	{attribute 'TcIecLibraryType'}
	{attribute 'external_name' := 'F_VN_GetAffineTransformation2D_GUID_6DC20EB8_D1ED_DF72_BBA8_AC231DAC2366'}
	(* Estimate the 2D affine transformation between two planar point sets using RANSAC algorithm. *)
	FUNCTION F_VN_GetAffineTransformation2D : HRESULT
	VAR_INPUT
		ipSrcPoints	:	ITcVnContainer;	(* Container with at least 3 source points (ContainerType_Vector_TcVnPoint2_REAL) *)
		ipDestPoints	:	ITcVnContainer;	(* Container with destination points (same number as ipSrcPoints, ContainerType_Vector_TcVnPoint2_REAL) *)
	END_VAR
	VAR_IN_OUT
		aAffineTransform	:	TcVnMatrix2x3_LREAL;	(* Returns the affine transformation matrix, which transforms the source points to the destination points *)
	END_VAR
	VAR_INPUT
		hrPrev	:	HRESULT;	(* HRESULT indicating the result of previous operations (If SUCCEEDED(hrPrev) equals false, no operation is executed.) *)
	END_VAR

END_FUNCTION

// Functions/Geometric and Coordinate Transformations/F_VN_GetAffineTransformation2DExp

	{attribute 'TcIecLibraryType'}
	{attribute 'external_name' := 'F_VN_GetAffineTransformation2DExp_GUID_BF2309E8_DA28_DC6D_B5BB_59115DF4FCE5'}
	(* Estimate the affine transformation between two planar point sets. (expert function) *)
	FUNCTION F_VN_GetAffineTransformation2DExp : HRESULT
	VAR_INPUT
		ipSrcPoints	:	ITcVnContainer;	(* Container with at least 3 source points (ContainerType_Vector_TcVnPoint2_REAL) *)
		ipDestPoints	:	ITcVnContainer;	(* Container with destination points (same number as ipSrcPoints, ContainerType_Vector_TcVnPoint2_REAL) *)
	END_VAR
	VAR_IN_OUT
		aAffineTransform	:	TcVnMatrix2x3_LREAL;	(* Returns the affine transformation matrix, which transforms the source points to the destination points *)
	END_VAR
	VAR_INPUT
		eAlgorithm	:	ETcVnEstimationAlgorithm;	(* Estimation algorithm (only RANSAC and LMEDS are supported) *)
		fReprojThreshold	:	LREAL;	(* Maximum allowed reprojection error to treat a point pair as an inlier *)
		ipInlierMask	:	REFERENCE TO ITcVnContainer;	(* Returns a mask marking the inliers (optional, set to 0 if not required; ContainerType_Vector_USINT) *)
		nMaxIterations	:	UDINT;	(* Maximum number of iterations *)
		fConfidence	:	LREAL;	(* Confidence (0..1) *)
		nRefineIters	:	UDINT;	(* Maximum number of iterations of Levenberg-Marquardt algorithm to refine further the affine transform (using only inliers). Set to 0 to disable refining. *)
		hrPrev	:	HRESULT;	(* HRESULT indicating the result of previous operations (If SUCCEEDED(hrPrev) equals false, no operation is executed.) *)
	END_VAR

END_FUNCTION

// Functions/Geometric and Coordinate Transformations/F_VN_GetPerspectiveTransformation

	{attribute 'TcIecLibraryType'}
	{attribute 'external_name' := 'F_VN_GetPerspectiveTransformation_GUID_EB7791C6_2E8A_D6F1_9211_DDA5AEA43AB7'}
	(* Calculate the perspective transformation between four corresponding point pairs. The points mark the corners of the corresponding rectangles. *)
	FUNCTION F_VN_GetPerspectiveTransformation : HRESULT
	VAR_IN_OUT
		aSrcPoints	:	TcVnArray4_Point2_REAL;	(* Source points *)
		aDestPoints	:	TcVnArray4_Point2_REAL;	(* Destination points *)
		aTransformationMatrix	:	TcVnMatrix3x3_LREAL;	(* Resulting transformation matrix *)
	END_VAR
	VAR_INPUT
		hrPrev	:	HRESULT;	(* HRESULT indicating the result of previous operations (If SUCCEEDED(hrPrev) equals false, no operation is executed.) *)
	END_VAR

END_FUNCTION

// Functions/Geometric and Coordinate Transformations/F_VN_Homography

	{attribute 'TcIecLibraryType'}
	{attribute 'external_name' := 'F_VN_Homography_GUID_95B7F292_17EB_D891_A27F_6BCFD1281378'}
	(* Find the homography (perspective transformation) between two planar point sets using RANSAC algorithm. *)
	FUNCTION F_VN_Homography : HRESULT
	VAR_INPUT
		ipSrcPoints	:	ITcVnContainer;	(* Container with at least 4 source points (ContainerType_Vector_TcVnPoint2_REAL) *)
		ipDestPoints	:	ITcVnContainer;	(* Container with destination points (same number as ipSrcPoints, ContainerType_Vector_TcVnPoint2_REAL) *)
	END_VAR
	VAR_IN_OUT
		aPerspectiveTransform	:	TcVnMatrix3x3_LREAL;	(* Returns the perspective transformation matrix, which transforms the source points to the destination points *)
	END_VAR
	VAR_INPUT
		hrPrev	:	HRESULT;	(* HRESULT indicating the result of previous operations (If SUCCEEDED(hrPrev) equals false, no operation is executed.) *)
	END_VAR

END_FUNCTION

// Functions/Geometric and Coordinate Transformations/F_VN_HomographyExp

	{attribute 'TcIecLibraryType'}
	{attribute 'external_name' := 'F_VN_HomographyExp_GUID_BA02E438_C093_D953_9D0D_2FEBD7581D2F'}
	(* Find the homography (perspective transformation) between two planar point sets. (expert function) *)
	FUNCTION F_VN_HomographyExp : HRESULT
	VAR_INPUT
		ipSrcPoints	:	ITcVnContainer;	(* Container with at least 4 source points (ContainerType_Vector_TcVnPoint2_REAL) *)
		ipDestPoints	:	ITcVnContainer;	(* Container with destination points (same number as ipSrcPoints, ContainerType_Vector_TcVnPoint2_REAL) *)
	END_VAR
	VAR_IN_OUT
		aPerspectiveTransform	:	TcVnMatrix3x3_LREAL;	(* Returns the perspective transformation matrix, which transforms the source points to the destination points *)
	END_VAR
	VAR_INPUT
		eAlgorithm	:	ETcVnEstimationAlgorithm;	(* Estimation algorithm *)
		fReprojThreshold	:	LREAL;	(* Maximum allowed reprojection error to treat a point pair as an inlier (only for RANSAC, RHO) *)
		ipInlierMask	:	REFERENCE TO ITcVnContainer;	(* Returns a mask marking the inliers (optional, set to 0 if not required; ContainerType_Vector_SINT; only for RANSAC, LMEDS) *)
		nMaxIterations	:	UDINT;	(* Maximum number of RANSAC iterations *)
		fConfidence	:	LREAL;	(* Confidence (0..1) *)
		hrPrev	:	HRESULT;	(* HRESULT indicating the result of previous operations (If SUCCEEDED(hrPrev) equals false, no operation is executed.) *)
	END_VAR

END_FUNCTION

// Functions/Geometric and Coordinate Transformations/F_VN_InvertAffineTransformation

	{attribute 'TcIecLibraryType'}
	{attribute 'external_name' := 'F_VN_InvertAffineTransformation_GUID_B3AA109D_1663_D0EB_9259_686F19B830A0'}
	(* Invert a 2D affine transformation matrix. The inverted transformation compensates the affine transformation on an image if it is used in the F_VN_WarpAffine function. *)
	FUNCTION F_VN_InvertAffineTransformation : HRESULT
	VAR_IN_OUT
		aTransformationMatrix	:	TcVnMatrix2x3_LREAL;	(* Source affine transformation matrix *)
		aInvertedTransformationMatrix	:	TcVnMatrix2x3_LREAL;	(* Resulting inverted affine transformation matrix *)
	END_VAR
	VAR_INPUT
		hrPrev	:	HRESULT;	(* HRESULT indicating the result of previous operations (If SUCCEEDED(hrPrev) equals false, no operation is executed.) *)
	END_VAR

END_FUNCTION

// Functions/Geometric and Coordinate Transformations/F_VN_WarpAffine

	{attribute 'TcIecLibraryType'}
	{attribute 'external_name' := 'F_VN_WarpAffine_GUID_087F32E0_F118_D48A_B2E2_893EC8B4B590'}
	(* Apply an affine transformation to an image. *)
	FUNCTION F_VN_WarpAffine : HRESULT
	VAR_INPUT
		ipSrcImage	:	ITcVnImage;	(* Source image *)
		ipDestImage	:	REFERENCE TO ITcVnImage;	(* Destination image (An appropriate image will be created if required.) *)
	END_VAR
	VAR_IN_OUT
		aTransformationMatrix	:	TcVnMatrix2x3_LREAL;	(* Affine transformation matrix *)
	END_VAR
	VAR_INPUT
		hrPrev	:	HRESULT;	(* HRESULT indicating the result of previous operations (If SUCCEEDED(hrPrev) equals false, no operation is executed.) *)
	END_VAR

END_FUNCTION

// Functions/Geometric and Coordinate Transformations/F_VN_PerspectiveTransformation

	{attribute 'TcIecLibraryType'}
	{attribute 'external_name' := 'F_VN_PerspectiveTransformation_GUID_8E72088F_82FC_D8DE_9EC7_83F2BF441E9C'}
	(* Apply a perspective transformation (rotation + translation, e.g. from extrinsic calibration) to 3D point coordinates. *)
	FUNCTION F_VN_PerspectiveTransformation : HRESULT
	VAR_INPUT
		ipSrcPoints	:	ITcVnContainer;	(* Container with 3D source points (TcVnPoint3_REAL or TcVnPoint3_LREAL) *)
		ipDestPoints	:	REFERENCE TO ITcVnContainer;	(* Returns the transformed points (same type as ipSrcPoints) *)
	END_VAR
	VAR_IN_OUT
		aRotationMatrix	:	TcVnMatrix3x3_LREAL;	(* 3x3 rotation matrix *)
		aTranslationVector	:	TcVnVector3_LREAL;	(* Translation vector *)
	END_VAR
	VAR_INPUT
		hrPrev	:	HRESULT;	(* HRESULT indicating the result of previous operations (If SUCCEEDED(hrPrev) equals false, no operation is executed.) *)
	END_VAR

END_FUNCTION

// Functions/Geometric and Coordinate Transformations/F_VN_PyramidDown

	{attribute 'TcIecLibraryType'}
	{attribute 'external_name' := 'F_VN_PyramidDown_GUID_8B15EA6D_4EA2_DA11_83A3_A2A8EAA19753'}
	(* Downsamples an image to half width and height. *)
	FUNCTION F_VN_PyramidDown : HRESULT
	VAR_INPUT
		ipSrcImage	:	ITcVnImage;	(* Source image *)
		ipDestImage	:	REFERENCE TO ITcVnImage;	(* Destination image (An appropriate destination image will be created if required.) *)
		hrPrev	:	HRESULT;	(* HRESULT indicating the result of previous operations (If SUCCEEDED(hrPrev) equals false, no operation is executed.) *)
	END_VAR

END_FUNCTION

// Functions/Geometric and Coordinate Transformations/F_VN_PyramidUp

	{attribute 'TcIecLibraryType'}
	{attribute 'external_name' := 'F_VN_PyramidUp_GUID_E81BEF84_D6CE_DC75_9B7A_122C5B883429'}
	(* Upsamples an image to double width and height. *)
	FUNCTION F_VN_PyramidUp : HRESULT
	VAR_INPUT
		ipSrcImage	:	ITcVnImage;	(* Source image *)
		ipDestImage	:	REFERENCE TO ITcVnImage;	(* Destination image (An appropriate destination image will be created if required.) *)
		hrPrev	:	HRESULT;	(* HRESULT indicating the result of previous operations (If SUCCEEDED(hrPrev) equals false, no operation is executed.) *)
	END_VAR

END_FUNCTION

// Functions/Geometric and Coordinate Transformations/F_VN_RemapImageToLogPolarSpace

	{attribute 'TcIecLibraryType'}
	{attribute 'external_name' := 'F_VN_RemapImageToLogPolarSpace_GUID_1E076C05_F39F_DDA1_AEBF_84A0AEDD278A'}
	(* Remap an image to log-polar space. *)
	FUNCTION F_VN_RemapImageToLogPolarSpace : HRESULT
	VAR_INPUT
		ipSrcImage	:	ITcVnImage;	(* Source image *)
		ipDestImage	:	REFERENCE TO ITcVnImage;	(* Destination image (Must not be the same as ipSrcImage! An appropriate destination image will be created if required.) *)
	END_VAR
	VAR_IN_OUT
		aCenter	:	TcVnPoint2_REAL;	(* Center point for the transformation *)
	END_VAR
	VAR_INPUT
		hrPrev	:	HRESULT;	(* HRESULT indicating the result of previous operations (If SUCCEEDED(hrPrev) equals false, no operation is executed.) *)
	END_VAR

END_FUNCTION

// Functions/Geometric and Coordinate Transformations/F_VN_RemapImageToLogPolarSpaceExp

	{attribute 'TcIecLibraryType'}
	{attribute 'external_name' := 'F_VN_RemapImageToLogPolarSpaceExp_GUID_EB2B1852_BFD3_DFEA_986A_C7676446261F'}
	(* Remap an image to log-polar space. (expert function) *)
	FUNCTION F_VN_RemapImageToLogPolarSpaceExp : HRESULT
	VAR_INPUT
		ipSrcImage	:	ITcVnImage;	(* Source image *)
		ipDestImage	:	REFERENCE TO ITcVnImage;	(* Destination image (Must not be the same as ipSrcImage! An appropriate destination image will be created if required.) *)
	END_VAR
	VAR_IN_OUT
		aCenter	:	TcVnPoint2_REAL;	(* Center point for the transformation *)
	END_VAR
	VAR_INPUT
		fScale	:	LREAL;	(* Magnitude scale parameter, i.e. image width / ln(radius) (set to 0 for auto select) *)
		eInterpolationType	:	ETcVnInterpolationType;	(* Interpolation type *)
		hrPrev	:	HRESULT;	(* HRESULT indicating the result of previous operations (If SUCCEEDED(hrPrev) equals false, no operation is executed.) *)
	END_VAR

END_FUNCTION

// Functions/Geometric and Coordinate Transformations/F_VN_RemapImageToLogPolarSpaceExp2

	{attribute 'TcIecLibraryType'}
	{attribute 'external_name' := 'F_VN_RemapImageToLogPolarSpaceExp2_GUID_A3D95464_1FCF_DA4B_BAB6_58B9B01AC040'}
	(* Remap an image to log-polar space. (expert function) *)
	FUNCTION F_VN_RemapImageToLogPolarSpaceExp2 : HRESULT
	VAR_INPUT
		ipSrcImage	:	ITcVnImage;	(* Source image *)
		ipDestImage	:	REFERENCE TO ITcVnImage;	(* Destination image (Must not be the same as ipSrcImage! An appropriate destination image will be created if required.) *)
	END_VAR
	VAR_IN_OUT
		aCenter	:	TcVnPoint2_REAL;	(* Center point for the transformation *)
	END_VAR
	VAR_INPUT
		fScale	:	LREAL;	(* Magnitude scale parameter, i.e. image width / ln(radius) (set to 0 for auto select) *)
		eInterpolationType	:	ETcVnInterpolationType;	(* Interpolation type *)
		nDestWidth	:	DINT;	(* Destination image width (set to -1 for source image width, 0 to auto scale to transformed radius, > 0 for a user defined width) *)
		nDestHeight	:	DINT;	(* destination image height (set to -1 for source image height, 0 to auto scale to transformed radius * PI, > 0 for a user defined height) *)
		hrPrev	:	HRESULT;	(* HRESULT indicating the result of previous operations (If SUCCEEDED(hrPrev) equals false, no operation is executed.) *)
	END_VAR

END_FUNCTION

// Functions/Geometric and Coordinate Transformations/F_VN_RemapImageToPolarSpace

	{attribute 'TcIecLibraryType'}
	{attribute 'external_name' := 'F_VN_RemapImageToPolarSpace_GUID_AEDB1598_FA72_D6F8_AFA2_9A39B196FC94'}
	(* Remap an image to polar space. *)
	FUNCTION F_VN_RemapImageToPolarSpace : HRESULT
	VAR_INPUT
		ipSrcImage	:	ITcVnImage;	(* Source image *)
		ipDestImage	:	REFERENCE TO ITcVnImage;	(* Destination image (Must not be the same as ipSrcImage! An appropriate destination image will be created if required.) *)
	END_VAR
	VAR_IN_OUT
		aCenter	:	TcVnPoint2_REAL;	(* Center point for the transformation *)
	END_VAR
	VAR_INPUT
		hrPrev	:	HRESULT;	(* HRESULT indicating the result of previous operations (If SUCCEEDED(hrPrev) equals false, no operation is executed.) *)
	END_VAR

END_FUNCTION

// Functions/Geometric and Coordinate Transformations/F_VN_RemapImageToPolarSpaceExp

	{attribute 'TcIecLibraryType'}
	{attribute 'external_name' := 'F_VN_RemapImageToPolarSpaceExp_GUID_E8FE08D5_A345_DFCC_B279_88644749BBBB'}
	(* Remap an image to polar space. (expert function) *)
	FUNCTION F_VN_RemapImageToPolarSpaceExp : HRESULT
	VAR_INPUT
		ipSrcImage	:	ITcVnImage;	(* Source image *)
		ipDestImage	:	REFERENCE TO ITcVnImage;	(* Destination image (Must not be the same as ipSrcImage! An appropriate destination image will be created if required.) *)
	END_VAR
	VAR_IN_OUT
		aCenter	:	TcVnPoint2_REAL;	(* Center point for the transformation *)
	END_VAR
	VAR_INPUT
		fMaxRadius	:	LREAL;	(* Maximum radius for the transformation (set to 0 for auto select) *)
		eInterpolationType	:	ETcVnInterpolationType;	(* Interpolation type *)
		hrPrev	:	HRESULT;	(* HRESULT indicating the result of previous operations (If SUCCEEDED(hrPrev) equals false, no operation is executed.) *)
	END_VAR

END_FUNCTION

// Functions/Geometric and Coordinate Transformations/F_VN_RemapImageToPolarSpaceExp2

	{attribute 'TcIecLibraryType'}
	{attribute 'external_name' := 'F_VN_RemapImageToPolarSpaceExp2_GUID_1395427E_D813_DEAA_A222_67CB032B0E27'}
	(* Remap an image to polar space. (expert function) *)
	FUNCTION F_VN_RemapImageToPolarSpaceExp2 : HRESULT
	VAR_INPUT
		ipSrcImage	:	ITcVnImage;	(* Source image *)
		ipDestImage	:	REFERENCE TO ITcVnImage;	(* Destination image (Must not be the same as ipSrcImage! An appropriate destination image will be created if required.) *)
	END_VAR
	VAR_IN_OUT
		aCenter	:	TcVnPoint2_REAL;	(* Center point for the transformation *)
	END_VAR
	VAR_INPUT
		fMaxRadius	:	LREAL;	(* Maximum radius for the transformation (set to 0 for auto select) *)
		eInterpolationType	:	ETcVnInterpolationType;	(* Interpolation type *)
		nDestWidth	:	DINT;	(* Destination image width (set to -1 for source image width, 0 to auto scale to transformed radius, > 0 for a user defined width) *)
		nDestHeight	:	DINT;	(* destination image height (set to -1 for source image height, 0 to auto scale to transformed radius * PI, > 0 for a user defined height) *)
		hrPrev	:	HRESULT;	(* HRESULT indicating the result of previous operations (If SUCCEEDED(hrPrev) equals false, no operation is executed.) *)
	END_VAR

END_FUNCTION

// Functions/Geometric and Coordinate Transformations/F_VN_ResizeImage

	{attribute 'TcIecLibraryType'}
	{attribute 'external_name' := 'F_VN_ResizeImage_GUID_9DEE2688_ACCD_D306_9087_D82853F9CD76'}
	(* Resize an image using a specific interpolation type. *)
	FUNCTION F_VN_ResizeImage : HRESULT
	VAR_INPUT
		ipSrcImage	:	ITcVnImage;	(* Source image *)
		ipDestImage	:	REFERENCE TO ITcVnImage;	(* Destination image (An appropriate image will be created if required.) *)
		nWidth	:	UDINT;	(* New width *)
		nHeight	:	UDINT;	(* New height *)
		eInterpolationType	:	ETcVnInterpolationType;	(* Interpolation type *)
		hrPrev	:	HRESULT;	(* HRESULT indicating the result of previous operations (If SUCCEEDED(hrPrev) equals false, no operation is executed.) *)
	END_VAR

END_FUNCTION

// Functions/Geometric and Coordinate Transformations/F_VN_ResizeImageExp

	{attribute 'TcIecLibraryType'}
	{attribute 'external_name' := 'F_VN_ResizeImageExp_GUID_47E9EB68_2546_D298_86DE_B25F7A66B172'}
	(* Resize an image using a specific interpolation type while maintaining its aspect ratio. (expert function) *)
	FUNCTION F_VN_ResizeImageExp : HRESULT
	VAR_INPUT
		ipSrcImage	:	ITcVnImage;	(* Source image *)
		ipDestImage	:	REFERENCE TO ITcVnImage;	(* Destination image (An appropriate image will be created if required.) *)
		nWidth	:	UDINT;	(* New width *)
		nHeight	:	UDINT;	(* New height *)
		eInterpolationType	:	ETcVnInterpolationType;	(* Interpolation type *)
		ePaddingMode	:	ETcVnPaddingMode;	(* Image padding mode *)
	END_VAR
	VAR_IN_OUT
		aBorderValue	:	TcVnVector4_LREAL;	(* Border value, if TCVN_PM_LETTERBOX is used *)
	END_VAR
	VAR_INPUT
		hrPrev	:	HRESULT;	(* HRESULT indicating the result of previous operations (If SUCCEEDED(hrPrev) equals false, no operation is executed.) *)
	END_VAR

END_FUNCTION

// Functions/Geometric and Coordinate Transformations/F_VN_RotateImage

	{attribute 'TcIecLibraryType'}
	{attribute 'external_name' := 'F_VN_RotateImage_GUID_FC35D73F_A7D7_D327_BFBB_869110D8E88B'}
	(* Rotate an image by 90, 180, or 270 degrees in clockwise direction. *)
	FUNCTION F_VN_RotateImage : HRESULT
	VAR_INPUT
		ipSrcImage	:	ITcVnImage;	(* Source image *)
		ipDestImage	:	REFERENCE TO ITcVnImage;	(* Destination image (An appropriate image will be created if required.) *)
		eAngle	:	ETcVnRotationAngle;	(* Rotation angle *)
		hrPrev	:	HRESULT;	(* HRESULT indicating the result of previous operations (If SUCCEEDED(hrPrev) equals false, no operation is executed.) *)
	END_VAR

END_FUNCTION

// Functions/Geometric and Coordinate Transformations/F_VN_RotateImageExp

	{attribute 'TcIecLibraryType'}
	{attribute 'external_name' := 'F_VN_RotateImageExp_GUID_D2BE97AC_2740_D405_86F9_A9287C8A7BD0'}
	(* Rotate an image by an individual rotation angle in degrees. *)
	FUNCTION F_VN_RotateImageExp : HRESULT
	VAR_INPUT
		ipSrcImage	:	ITcVnImage;	(* Source image *)
		ipDestImage	:	REFERENCE TO ITcVnImage;	(* Destination image (An appropriate image will be created if required.) *)
		fAngleDeg	:	LREAL;	(* Rotation angle in degree (positive: counter-clockwise, negative: clockwise) *)
		bAdjustDestSize	:	BOOL;	(* If true, ipDestImage size is adjusted so that the whole rotated ipSrcImage is contained. Otherwise, ipDestImage size is set to ipSrcImage size. *)
		hrPrev	:	HRESULT;	(* HRESULT indicating the result of previous operations (If SUCCEEDED(hrPrev) equals false, no operation is executed.) *)
	END_VAR

END_FUNCTION

// Functions/Geometric and Coordinate Transformations/F_VN_RotateImageExp2

	{attribute 'TcIecLibraryType'}
	{attribute 'external_name' := 'F_VN_RotateImageExp2_GUID_F56926A3_8407_DE46_8D68_B89F032FA20A'}
	(* Rotate an image by an individual rotation angle in degrees. (expert function) *)
	FUNCTION F_VN_RotateImageExp2 : HRESULT
	VAR_INPUT
		ipSrcImage	:	ITcVnImage;	(* Source image *)
		ipDestImage	:	REFERENCE TO ITcVnImage;	(* Destination image (An appropriate image will be created if required.) *)
		fAngleDeg	:	LREAL;	(* Rotation angle in degree (positive: counter-clockwise, negative: clockwise) *)
		bAdjustDestSize	:	BOOL;	(* If true, ipDestImage size is adjusted so that the whole rotated ipSrcImage is contained. Otherwise, ipDestImage size is set to ipSrcImage size. *)
		eInterpolationType	:	ETcVnInterpolationType;	(* Interpolation method *)
		eBorderInterpolation	:	ETcVnBorderInterpolationMethod;	(* Border interpolation method (ISOLATED not supported) *)
	END_VAR
	VAR_IN_OUT
		aBorderValue	:	TcVnVector4_LREAL;	(* Border value, if CONSTANT is used *)
	END_VAR
	VAR_INPUT
		hrPrev	:	HRESULT;	(* HRESULT indicating the result of previous operations (If SUCCEEDED(hrPrev) equals false, no operation is executed.) *)
	END_VAR

END_FUNCTION

// Functions/Geometric and Coordinate Transformations/F_VN_WarpAffineExp

	{attribute 'TcIecLibraryType'}
	{attribute 'external_name' := 'F_VN_WarpAffineExp_GUID_95552B05_373D_D85A_A644_4CE2C5CCCE45'}
	(* Apply an affine transformation to an image. (expert function) *)
	FUNCTION F_VN_WarpAffineExp : HRESULT
	VAR_INPUT
		ipSrcImage	:	ITcVnImage;	(* Source image *)
		ipDestImage	:	REFERENCE TO ITcVnImage;	(* Destination image (An appropriate image will be created if required.) *)
	END_VAR
	VAR_IN_OUT
		aTransformationMatrix	:	TcVnMatrix2x3_LREAL;	(* Affine transformation matrix *)
	END_VAR
	VAR_INPUT
		nDestWidth	:	UDINT;	(* Width of the destination image *)
		nDestHeight	:	UDINT;	(* Height of the destination image *)
		eInterpolationType	:	ETcVnInterpolationType;	(* Interpolation method *)
		bWarpInverse	:	BOOL;	(* Handle aTransformationMatrix as the inverse transformation *)
		eBorderInterpolation	:	ETcVnBorderInterpolationMethod;	(* Border interpolation method (ISOLATED not supported) *)
		fBorderValue	:	LREAL;	(* Border value, if CONSTANT is used *)
		hrPrev	:	HRESULT;	(* HRESULT indicating the result of previous operations (If SUCCEEDED(hrPrev) equals false, no operation is executed.) *)
	END_VAR

END_FUNCTION

// Functions/Geometric and Coordinate Transformations/F_VN_WarpAffine_Container

	{attribute 'TcIecLibraryType'}
	{attribute 'external_name' := 'F_VN_WarpAffine_Container_GUID_CD3C3C3B_4C4A_DAE7_93B8_C3EE1865484A'}
	(* Apply an affine transformation to a container of 2D points. *)
	FUNCTION F_VN_WarpAffine_Container : HRESULT
	VAR_INPUT
		ipSrcPoints	:	ITcVnContainer;	(* Source points (ContainerType_Vector_TcVnPoint2_DINT or ContainerType_Vector_TcVnPoint2_REAL or ContainerType_Vector_TcVnPoint2_LREAL) *)
		ipDestPoints	:	REFERENCE TO ITcVnContainer;	(* Returns the transformed points (same type ID as ipSrcPoints; Non-zero interface pointers are reused.) *)
	END_VAR
	VAR_IN_OUT
		aTransformationMatrix	:	TcVnMatrix2x3_LREAL;	(* Affine transformation matrix *)
	END_VAR
	VAR_INPUT
		hrPrev	:	HRESULT;	(* HRESULT indicating the result of previous operations (If SUCCEEDED(hrPrev) equals false, no operation is executed.) *)
	END_VAR

END_FUNCTION

// Functions/Geometric and Coordinate Transformations/F_VN_WarpAffine_Point

	{attribute 'TcIecLibraryType'}
	{attribute 'external_name' := 'F_VN_WarpAffine_Point_GUID_7CFB431B_7051_DF9F_AFCD_02E59F0F9818'}
	(* Apply an affine transformation to a 2D point. *)
	FUNCTION F_VN_WarpAffine_Point : HRESULT
	VAR_IN_OUT
		aSrcPoint	:	TcVnPoint2_LREAL;	(* Source point *)
		aDestPoint	:	TcVnPoint2_LREAL;	(* Destination point *)
		aTransformationMatrix	:	TcVnMatrix2x3_LREAL;	(* Affine transformation matrix *)
	END_VAR
	VAR_INPUT
		hrPrev	:	HRESULT;	(* HRESULT indicating the result of previous operations (If SUCCEEDED(hrPrev) equals false, no operation is executed.) *)
	END_VAR

END_FUNCTION

// Functions/Geometric and Coordinate Transformations/F_VN_WarpAffine_Rectangle

	{attribute 'TcIecLibraryType'}
	{attribute 'external_name' := 'F_VN_WarpAffine_Rectangle_GUID_2C93C147_3D1A_DCEC_A8D2_2F0EE7AA65E1'}
	(* Use an affine transform to warp a rectangle. *)
	FUNCTION F_VN_WarpAffine_Rectangle : HRESULT
	VAR_INPUT
		nTopLeftX	:	UDINT;	(* x coordinate of the top left corner *)
		nTopLeftY	:	UDINT;	(* y coordinate of the top left corner *)
		nBottomRightX	:	UDINT;	(* x coordinate of the bottom right corner *)
		nBottomRightY	:	UDINT;	(* y coordinate of the bottom right corner *)
		ipDestPoints	:	REFERENCE TO ITcVnContainer;	(* Returns the 4 transformed points (ContainerType_Vector_TcVnPoint2_REAL) *)
	END_VAR
	VAR_IN_OUT
		aTransformationMatrix	:	TcVnMatrix2x3_LREAL;	(* Affine transformation matrix *)
	END_VAR
	VAR_INPUT
		hrPrev	:	HRESULT;	(* HRESULT indicating the result of previous operations (If SUCCEEDED(hrPrev) equals false, no operation is executed.) *)
	END_VAR

END_FUNCTION

// Functions/Geometric and Coordinate Transformations/F_VN_WarpPerspective

	{attribute 'TcIecLibraryType'}
	{attribute 'external_name' := 'F_VN_WarpPerspective_GUID_8AC97FBA_4792_D990_BFB6_F503396FB2B9'}
	(* Apply a perspective transformation to an image. *)
	FUNCTION F_VN_WarpPerspective : HRESULT
	VAR_INPUT
		ipSrcImage	:	ITcVnImage;	(* Source image *)
		ipDestImage	:	REFERENCE TO ITcVnImage;	(* Destination image (An appropriate image will be created if required.) *)
	END_VAR
	VAR_IN_OUT
		aTransformationMatrix	:	TcVnMatrix3x3_LREAL;	(* Perspective transformation matrix *)
	END_VAR
	VAR_INPUT
		hrPrev	:	HRESULT;	(* HRESULT indicating the result of previous operations (If SUCCEEDED(hrPrev) equals false, no operation is executed.) *)
	END_VAR

END_FUNCTION

// Functions/Geometric and Coordinate Transformations/F_VN_WarpPerspective_Container

	{attribute 'TcIecLibraryType'}
	{attribute 'external_name' := 'F_VN_WarpPerspective_Container_GUID_811C143E_6004_D660_998A_A4D4DDC19A5B'}
	(* Apply a perspective transformation to a container of 2D points. *)
	FUNCTION F_VN_WarpPerspective_Container : HRESULT
	VAR_INPUT
		ipSrcPoints	:	ITcVnContainer;	(* Source points (ContainerType_Vector_TcVnPoint2_DINT or ContainerType_Vector_TcVnPoint2_REAL or ContainerType_Vector_TcVnPoint2_LREAL) *)
		ipDestPoints	:	REFERENCE TO ITcVnContainer;	(* Returns the transformed points (same type ID as ipSrcPoints; Non-zero interface pointers are reused.) *)
	END_VAR
	VAR_IN_OUT
		aTransformationMatrix	:	TcVnMatrix3x3_LREAL;	(* Perspective transformation matrix *)
	END_VAR
	VAR_INPUT
		hrPrev	:	HRESULT;	(* HRESULT indicating the result of previous operations (If SUCCEEDED(hrPrev) equals false, no operation is executed.) *)
	END_VAR

END_FUNCTION

// Functions/Geometric and Coordinate Transformations/F_VN_WarpPerspectiveExp

	{attribute 'TcIecLibraryType'}
	{attribute 'external_name' := 'F_VN_WarpPerspectiveExp_GUID_719F5D10_97B4_DC85_AAFF_3AEC5320AF57'}
	(* Apply a perspective transformation to an image. (expert function) *)
	FUNCTION F_VN_WarpPerspectiveExp : HRESULT
	VAR_INPUT
		ipSrcImage	:	ITcVnImage;	(* Source image *)
		ipDestImage	:	REFERENCE TO ITcVnImage;	(* Destination image (An appropriate image will be created if required.) *)
	END_VAR
	VAR_IN_OUT
		aTransformationMatrix	:	TcVnMatrix3x3_LREAL;	(* Perspective transformation matrix *)
	END_VAR
	VAR_INPUT
		nDestWidth	:	UDINT;	(* Width of the destination image *)
		nDestHeight	:	UDINT;	(* Height of the destination image *)
		eInterpolationType	:	ETcVnInterpolationType;	(* Interpolation method *)
		bWarpInverse	:	BOOL;	(* Handle aTransformationMatrix as the inverse transformation *)
		eBorderInterpolation	:	ETcVnBorderInterpolationMethod;	(* Border interpolation method (ISOLATED not supported) *)
		fBorderValue	:	LREAL;	(* Border value, if CONSTANT is used *)
		hrPrev	:	HRESULT;	(* HRESULT indicating the result of previous operations (If SUCCEEDED(hrPrev) equals false, no operation is executed.) *)
	END_VAR

END_FUNCTION

// Functions/Geometric and Coordinate Transformations/F_VN_WarpPerspective_Point

	{attribute 'TcIecLibraryType'}
	{attribute 'external_name' := 'F_VN_WarpPerspective_Point_GUID_7A416256_BFE9_DE26_B5CC_C06151EF0391'}
	(* Apply a perspective transformation to a 2D point. *)
	FUNCTION F_VN_WarpPerspective_Point : HRESULT
	VAR_IN_OUT
		aSrcPoint	:	TcVnPoint2_LREAL;	(* Source point *)
		aDestPoint	:	TcVnPoint2_LREAL;	(* Destination point *)
		aTransformationMatrix	:	TcVnMatrix3x3_LREAL;	(* Perspective transformation matrix *)
	END_VAR
	VAR_INPUT
		hrPrev	:	HRESULT;	(* HRESULT indicating the result of previous operations (If SUCCEEDED(hrPrev) equals false, no operation is executed.) *)
	END_VAR

END_FUNCTION

// Functions/Geometric and Coordinate Transformations/F_VN_WarpPerspective_Rectangle

	{attribute 'TcIecLibraryType'}
	{attribute 'external_name' := 'F_VN_WarpPerspective_Rectangle_GUID_8C2C5CDD_5FD1_DA1C_AE6F_8DE3FF646238'}
	(* Use a perspective transform to warp a rectangle. *)
	FUNCTION F_VN_WarpPerspective_Rectangle : HRESULT
	VAR_INPUT
		nTopLeftX	:	UDINT;	(* x coordinate of the top left corner *)
		nTopLeftY	:	UDINT;	(* y coordinate of the top left corner *)
		nBottomRightX	:	UDINT;	(* x coordinate of the bottom right corner *)
		nBottomRightY	:	UDINT;	(* y coordinate of the bottom right corner *)
		ipDestPoints	:	REFERENCE TO ITcVnContainer;	(* Returns the 4 transformed points (ContainerType_Vector_TcVnPoint2_REAL) *)
	END_VAR
	VAR_IN_OUT
		aTransformationMatrix	:	TcVnMatrix3x3_LREAL;	(* Perspective transformation matrix *)
	END_VAR
	VAR_INPUT
		hrPrev	:	HRESULT;	(* HRESULT indicating the result of previous operations (If SUCCEEDED(hrPrev) equals false, no operation is executed.) *)
	END_VAR

END_FUNCTION

// Functions/Image Color and Contrast Processing/F_VN_ApplyColorMap

	{attribute 'TcIecLibraryType'}
	{attribute 'external_name' := 'F_VN_ApplyColorMap_GUID_1AED99AE_B422_DB03_B79D_6AF5C816ED50'}
	(* Apply a color map to a gray-level image. *)
	FUNCTION F_VN_ApplyColorMap : HRESULT
	VAR_INPUT
		ipSrcImage	:	ITcVnImage;	(* Source image (TCVN_ET_USINT or TCVN_ET_UINT, 1 channel) *)
		ipDestImage	:	REFERENCE TO ITcVnImage;	(* Returns the colored image (TCVN_ET_USINT, 3 channel. An appropriate image will be created if required.) *)
		ipColorMap	:	ITcVnContainer;	(* Color map to be applied to ipSrcImage (ContainerType_Vector_TcVnVector3_REAL with 256 or 65536 elements, dependent on ipSrcImage type). Can be either custom or created with F_VN_GenerateColorMap. *)
		hrPrev	:	HRESULT;	(* HRESULT indicating the result of previous operations (If SUCCEEDED(hrPrev) equals false, no operation is executed.) *)
	END_VAR

END_FUNCTION

// Functions/Image Color and Contrast Processing/F_VN_GenerateColorMap

	{attribute 'TcIecLibraryType'}
	{attribute 'external_name' := 'F_VN_GenerateColorMap_GUID_043E26EE_8DE2_D26C_9CCE_1A63D6E6F7D7'}
	(* Generates a pre-defined color map. *)
	FUNCTION F_VN_GenerateColorMap : HRESULT
	VAR_INPUT
		ipColorMap	:	REFERENCE TO ITcVnContainer;	(* Returns the color map (ContainerType_Vector_TcVnVector3_REAL with 256 or 65536 elements) *)
		eColorMap	:	ETcVnColorMap;	(* Selects a color map (similar to GNU Octave/MATLAB types) *)
		eColorMapSize	:	ETcVnColorMapSize;	(* Defines how many elements the generated color map should have *)
		hrPrev	:	HRESULT;	(* HRESULT indicating the result of previous operations (If SUCCEEDED(hrPrev) equals false, no operation is executed.) *)
	END_VAR

END_FUNCTION

// Functions/Image Color and Contrast Processing/F_VN_ApplyLut

	{attribute 'TcIecLibraryType'}
	{attribute 'external_name' := 'F_VN_ApplyLut_GUID_185F14D8_273A_DF28_B84D_07B552E99C4E'}
	(* Apply a lookup table to an image to manipulate its colors. *)
	FUNCTION F_VN_ApplyLut : HRESULT
	VAR_INPUT
		ipSrcImage	:	ITcVnImage;	(* Source image (1-4 channels of 8 or 16 bit types SINT, USINT, INT, UINT) *)
		ipDestImage	:	REFERENCE TO ITcVnImage;	(* Returns the result image (same size, type and channels as ipSrcImage. An appropriate image will be created if required.) *)
		ipLut	:	ITcVnContainer;	(* Lookup table with elements matching ipSrcImage type and either 256 (8 bit images) or 65536 (16 bit images) elements. E.g. ContainerType_Vector_USINT for 1-4 channel USINT image (in this case, the same lookup values are used for each channel) or ContainerType_Vector_TcVnVector3_USINT for a 3 channel USINT image (in this case, each channel uses an individual lookup value).
						 *)
		hrPrev	:	HRESULT;	(* HRESULT indicating the result of previous operations (If SUCCEEDED(hrPrev) equals false, no operation is executed.) *)
	END_VAR

END_FUNCTION

// Functions/Image Color and Contrast Processing/F_VN_Clahe

	{attribute 'TcIecLibraryType'}
	{attribute 'external_name' := 'F_VN_Clahe_GUID_2ABEF4E8_FD47_D68E_8F45_12C11E74C580'}
	(* Apply Constrast Limited Adaptive Histogram Equalization. This applies local histogram equalization to individual tiles. *)
	FUNCTION F_VN_Clahe : HRESULT
	VAR_INPUT
		ipSrcImage	:	ITcVnImage;	(* Source image (TCVN_ET_USINT or TCVN_ET_UINT, 1 channel) *)
		ipDestImage	:	REFERENCE TO ITcVnImage;	(* Returns the resulting image (An appropriate image will be created if required.) *)
		hrPrev	:	HRESULT;	(* HRESULT indicating the result of previous operations (If SUCCEEDED(hrPrev) equals false, no operation is executed.) *)
	END_VAR

END_FUNCTION

// Functions/Image Color and Contrast Processing/F_VN_ClaheExp

	{attribute 'TcIecLibraryType'}
	{attribute 'external_name' := 'F_VN_ClaheExp_GUID_9082C14A_966D_D6E8_B339_52E6FEA896AE'}
	(* Apply Constrast Limited Adaptive Histogram Equalization. This applies local histogram equalization to individual tiles. (expert function) *)
	FUNCTION F_VN_ClaheExp : HRESULT
	VAR_INPUT
		ipSrcImage	:	ITcVnImage;	(* Source image (TCVN_ET_USINT or TCVN_ET_UINT, 1 channel) *)
		ipDestImage	:	REFERENCE TO ITcVnImage;	(* Returns the resulting image (An appropriate image will be created if required.) *)
		fClipLimit	:	LREAL;	(* Threshold for contrast limit (set to <= 0 to disable clipping) *)
		nTilesX	:	UDINT;	(* Number of tiles in x direction *)
		nTilesY	:	UDINT;	(* Number of tiles in y direction *)
		hrPrev	:	HRESULT;	(* HRESULT indicating the result of previous operations (If SUCCEEDED(hrPrev) equals false, no operation is executed.) *)
	END_VAR

END_FUNCTION

// Functions/Image Color and Contrast Processing/F_VN_ConvertColorSpace

	{attribute 'TcIecLibraryType'}
	{attribute 'external_name' := 'F_VN_ConvertColorSpace_GUID_7C0481CB_BD98_DFF7_BBC8_AFD17A257B54'}
	(* Convert image from one color space to another. *)
	FUNCTION F_VN_ConvertColorSpace : HRESULT
	VAR_INPUT
		ipSrcImage	:	ITcVnImage;	(* Source image *)
		ipDestImage	:	REFERENCE TO ITcVnImage;	(* Destination image (An appropriate destination image will be created if required.) *)
		eTransform	:	ETcVnColorSpaceTransform;	(* Transforms to be applied *)
		hrPrev	:	HRESULT;	(* HRESULT indicating the result of previous operations (If SUCCEEDED(hrPrev) equals false, no operation is executed.) *)
	END_VAR

END_FUNCTION

// Functions/Image Color and Contrast Processing/F_VN_GenerateCustomColorMap

	{attribute 'TcIecLibraryType'}
	{attribute 'external_name' := 'F_VN_GenerateCustomColorMap_GUID_600A3840_368F_D246_8D52_D3DE77BDD2D0'}
	(* Generate a custom color map by interpolating between user defined colors (equally distributed, linear for each channel). *)
	FUNCTION F_VN_GenerateCustomColorMap : HRESULT
	VAR_INPUT
		ipColorMap	:	REFERENCE TO ITcVnContainer;	(* Returns the color map (ContainerType_Vector_TcVnVector3_REAL with 256 or 65536 elements) *)
		ipInitialColors	:	ITcVnContainer;	(* User defined colors (ContainerType_Vector_TcVnVector3_REAL, at least 2 elements) *)
		eColorMapSize	:	ETcVnColorMapSize;	(* Defines how many elements the generated color map should have *)
		hrPrev	:	HRESULT;	(* HRESULT indicating the result of previous operations (If SUCCEEDED(hrPrev) equals false, no operation is executed.) *)
	END_VAR

END_FUNCTION

// Functions/Image Color and Contrast Processing/F_VN_Histogram

	{attribute 'TcIecLibraryType'}
	{attribute 'external_name' := 'F_VN_Histogram_GUID_0C4BC7AC_935E_D288_ADFA_C39F46FA9470'}
	(* Calculate the (multi-channel) histogram of an image. *)
	FUNCTION F_VN_Histogram : HRESULT
	VAR_INPUT
		ipSrcImage	:	ITcVnImage;	(* Source image *)
		ipDestHistogram	:	REFERENCE TO ITcVnContainer;	(* Returns a container with a multi-channel histogram, where every channel is represented as a vector of UDINT (ContainerType_Vector_Vector_UDINT. Non-zero interface pointers are reused.) *)
		hrPrev	:	HRESULT;	(* HRESULT indicating the result of previous operations (If SUCCEEDED(hrPrev) equals false, no operation is executed.) *)
	END_VAR

END_FUNCTION

// Functions/Image Color and Contrast Processing/F_VN_HistogramExp

	{attribute 'TcIecLibraryType'}
	{attribute 'external_name' := 'F_VN_HistogramExp_GUID_8761A615_7D31_D5FF_8B2D_AEBA565F0E28'}
	(* Calculate the (multi-channel) histogram of an image. (expert function) *)
	FUNCTION F_VN_HistogramExp : HRESULT
	VAR_INPUT
		ipSrcImage	:	ITcVnImage;	(* Source image *)
		ipDestHistogram	:	REFERENCE TO ITcVnContainer;	(* Returns a container with a multi-channel histogram, where every channel is represented as a vector of UDINT (ContainerType_Vector_Vector_UDINT. Non-zero interface pointers are reused.) *)
	END_VAR
	VAR_IN_OUT
		nBins	:	UDINT;	(* Desired number of bins or 0 to keep the default for the corresponding image format (in) and default number of bins (out) *)
		fLowerBound	:	LREAL;	(* Lower (inclusive) boundary of the 0-th histogram bin (in), or receive the default if fLowerBound AND fUpperBound are set to 0 (out) *)
		fUpperBound	:	LREAL;	(* Upper (exclusive) boundary of the last histogram bin nBins-1 (in), or receive the default if fLowerBound AND fUpperBound are set to 0 (out) *)
	END_VAR
	VAR_INPUT
		ipMask	:	ITcVnImage;	(* Source image mask (TCVN_ET_USINT, 1 channel. Mask is optional, set to 0 if not required.) *)
		hrPrev	:	HRESULT;	(* HRESULT indicating the result of previous operations (If SUCCEEDED(hrPrev) equals false, no operation is executed.) *)
	END_VAR

END_FUNCTION

// Functions/Image Color and Contrast Processing/F_VN_HistogramEqualization

	{attribute 'TcIecLibraryType'}
	{attribute 'external_name' := 'F_VN_HistogramEqualization_GUID_A18B75DF_31AC_D722_B696_230E6220D545'}
	(* Equalize the histogram of a grayscale or rgb image, which normalizes the brightness and improves the contrast. *)
	FUNCTION F_VN_HistogramEqualization : HRESULT
	VAR_INPUT
		ipSrcImage	:	ITcVnImage;	(* Source image (USINT) *)
		ipDestImage	:	REFERENCE TO ITcVnImage;	(* Destination image (An appropriate destination image will be created if required.) *)
		hrPrev	:	HRESULT;	(* HRESULT indicating the result of previous operations (If SUCCEEDED(hrPrev) equals false, no operation is executed.) *)
	END_VAR

END_FUNCTION

// Functions/Image Color and Contrast Processing/F_VN_HistogramEqualizationExp

	{attribute 'TcIecLibraryType'}
	{attribute 'external_name' := 'F_VN_HistogramEqualizationExp_GUID_CB98AC95_CB67_D82A_9BFD_5CE805561873'}
	(* Equalize the histogram of a grayscale or color image, which normalizes the brightness and improves the contrast. (expert function) 
	The channel index that should be equalized has to be specified (-1 expects a RGB image, converts it to YCbCr, equalizes the Y channel and converts the image back to RGB).  *)
	FUNCTION F_VN_HistogramEqualizationExp : HRESULT
	VAR_INPUT
		ipSrcImage	:	ITcVnImage;	(* Source image (USINT) *)
		ipDestImage	:	REFERENCE TO ITcVnImage;	(* Destination image (An appropriate destination image will be created if required.) *)
		nChannelIdx	:	INT;	(* Index of the image channel that should be equalized (-1 expects a RGB image, converts it to YCbCr, equalizes the Y channel and converts the image back to RGB) *)
		hrPrev	:	HRESULT;	(* HRESULT indicating the result of previous operations (If SUCCEEDED(hrPrev) equals false, no operation is executed.) *)
	END_VAR

END_FUNCTION

// Functions/Image Color and Contrast Processing/F_VN_InvertImageColor

	{attribute 'TcIecLibraryType'}
	{attribute 'external_name' := 'F_VN_InvertImageColor_GUID_729059A7_AEDC_D8E6_B8DC_22D18874C758'}
	(* Invert the color of an image.
          For signed integer or negative floating point values, only the signs will be switched.
          If the image contains only positive floating point values, each pixel value is subtracted from the maximum available pixel value (or 1.0, whatever is higher). *)
	FUNCTION F_VN_InvertImageColor : HRESULT
	VAR_INPUT
		ipSrcImage	:	ITcVnImage;	(* Source image *)
		ipDestImage	:	REFERENCE TO ITcVnImage;	(* Destination image (An appropriate image will be created if required.) *)
		hrPrev	:	HRESULT;	(* HRESULT indicating the result of previous operations (If SUCCEEDED(hrPrev) equals false, no operation is executed.) *)
	END_VAR

END_FUNCTION

// Functions/Image Color and Contrast Processing/F_VN_InvertImageColorExp

	{attribute 'TcIecLibraryType'}
	{attribute 'external_name' := 'F_VN_InvertImageColorExp_GUID_9DE64ABD_CFE4_D84C_8B93_7E3E2DF00694'}
	(* Invert the color of an image. (expert function)
          For signed integer or negative floating point values, only the signs will be switched.
          If the image contains only positive floating point values, each pixel value is subtracted from the maximum available pixel value (or 1.0, whatever is higher). *)
	FUNCTION F_VN_InvertImageColorExp : HRESULT
	VAR_INPUT
		ipSrcImage	:	ITcVnImage;	(* Source image *)
		ipDestImage	:	REFERENCE TO ITcVnImage;	(* Destination image (An appropriate image will be created if required.) *)
		fMaxValue	:	LREAL;	(* Maximum pixel value (e.g. if a 16 bit image contains 12 bit values). -1 means the default values are used. *)
		hrPrev	:	HRESULT;	(* HRESULT indicating the result of previous operations (If SUCCEEDED(hrPrev) equals false, no operation is executed.) *)
	END_VAR

END_FUNCTION

// Functions/Image Color and Contrast Processing/F_VN_NormalizeImage

	{attribute 'TcIecLibraryType'}
	{attribute 'external_name' := 'F_VN_NormalizeImage_GUID_44E520D2_4F74_D94C_8297_1C0D9D71CEC0'}
	(* Normalize an image regarding its value range (e.g. stretch pixel values [50..150] to full range [0..255]). *)
	FUNCTION F_VN_NormalizeImage : HRESULT
	VAR_INPUT
		ipSrcImage	:	ITcVnImage;	(* Source image *)
		ipDestImage	:	REFERENCE TO ITcVnImage;	(* Destination image (An appropriate destination image will be created if required.) *)
		hrPrev	:	HRESULT;	(* HRESULT indicating the result of previous operations (If SUCCEEDED(hrPrev) equals false, no operation is executed.) *)
	END_VAR

END_FUNCTION

// Functions/Image Color and Contrast Processing/F_VN_NormalizeImageExp

	{attribute 'TcIecLibraryType'}
	{attribute 'external_name' := 'F_VN_NormalizeImageExp_GUID_BC09673E_0A38_DCC6_A786_BA00F94A148C'}
	(* Normalize an image regarding its value range (e.g. stretch pixel values [50..150] to full range [0..255]) or scale the values regarding a specific normalization (e.g. L2-norm). (expert function) *)
	FUNCTION F_VN_NormalizeImageExp : HRESULT
	VAR_INPUT
		ipSrcImage	:	ITcVnImage;	(* Source image *)
		ipDestImage	:	REFERENCE TO ITcVnImage;	(* Destination image (An appropriate destination image will be created if required.) *)
		fAlpha	:	LREAL;	(* Lower range boundary (in case of normalizing the value range) or value to normalize to (||ipDestImage|| = fAlpha) *)
		fBeta	:	LREAL;	(* Upper range boundary (in case of normalizing the value range) *)
		eNormType	:	ETcVnNormalizationType;	(* Normalization type (only INF, L1, L2 or MINMAX) *)
		eDestType	:	ETcVnElementType;	(* Destination image depth (usually SAME_AS_SOURCE) *)
		ipMask	:	ITcVnImage;	(* Mask to restrict the normalization to specific pixel positions (set 0 to normalize the whole image) *)
		hrPrev	:	HRESULT;	(* HRESULT indicating the result of previous operations (If SUCCEEDED(hrPrev) equals false, no operation is executed.) *)
	END_VAR

END_FUNCTION

// Functions/Image Color and Contrast Processing/F_VN_NormalizeImageForDisplay

	{attribute 'TcIecLibraryType'}
	{attribute 'external_name' := 'F_VN_NormalizeImageForDisplay_GUID_1F15C351_80B6_D511_8524_747374CF3D5E'}
	(* Normalize an image for display, i.e. scale it to the full value range of the underlying data type (-1 to 1 for floating point). *)
	FUNCTION F_VN_NormalizeImageForDisplay : HRESULT
	VAR_INPUT
		ipSrcImage	:	ITcVnImage;	(* Source image *)
		ipDestImage	:	REFERENCE TO ITcVnImage;	(* Destination image (An appropriate destination image will be created if required.) *)
		eSignedNormalization	:	ETcVnSignedNormalization;	(* Option for normalizing signed values *)
		hrPrev	:	HRESULT;	(* HRESULT indicating the result of previous operations (If SUCCEEDED(hrPrev) equals false, no operation is executed.) *)
	END_VAR

END_FUNCTION

// Functions/Image Color and Contrast Processing/F_VN_ReferenceColorSimilarity_ITcVnColorModel

	{attribute 'TcIecLibraryType'}
	{attribute 'external_name' := 'F_VN_ReferenceColorSimilarity_ITcVnColorModel_GUID_6F33160A_281E_DC56_BDF2_4AA2317FC9D3'}
	(* Computes the similarity to a reference color model for each pixel in the source image. *)
	FUNCTION F_VN_ReferenceColorSimilarity_ITcVnColorModel : HRESULT
	VAR_INPUT
		ipSrcImage	:	ITcVnImage;	(* RGB source image (USINT, 3 channels) *)
		ipDestImage	:	REFERENCE TO ITcVnImage;	(* Returns the similarity to ipColorModel for each pixel in ipSrcImage (USINT, 1 channel. An appropriate destination image will be created if required.) *)
		ipColorModel	:	ITcVnColorModel;	(* Color model *)
		hrPrev	:	HRESULT;	(* HRESULT indicating the result of previous operations (If SUCCEEDED(hrPrev) equals false, no operation is executed.) *)
	END_VAR

END_FUNCTION

// Interfaces/Machine Learning/ITcVnColorModel

	(* Interface to train and classify an image color. *)
	{attribute 'c++_compatible'}
	{attribute 'vtable_order' := 'TrainImageColor;ClassifyImageColor'}
	INTERFACE ITcVnColorModel EXTENDS ITcVnMlModel


(* Train the color of the provided image. *)
	{attribute 'c++_compatible'}
	{attribute 'minimal_input_size' := '4'}
	{attribute 'pack_mode' := '4'}
	METHOD TrainImageColor : HRESULT
	VAR_INPUT
		ipSrcImage : ITcVnImage;
		nDifferentColors : UDINT;
		ipMask : ITcVnImage;
		nSkipPixels : UDINT;
	END_VAR
END_METHOD


(* Compute the similarity of each image pixel to the trained reference color. *)
	{attribute 'c++_compatible'}
	{attribute 'minimal_input_size' := '4'}
	{attribute 'pack_mode' := '4'}
	METHOD ClassifyImageColor : HRESULT
	VAR_INPUT
		ipSrcImage : ITcVnImage;
		pipDestImage : POINTER TO ITcVnImage;
		fVariance : REAL;
		fLuminanceWeight : REAL;
	END_VAR
END_METHOD

END_INTERFACE

// Functions/Image Color and Contrast Processing/F_VN_ReferenceColorSimilarityExp_ITcVnColorModel

	{attribute 'TcIecLibraryType'}
	{attribute 'external_name' := 'F_VN_ReferenceColorSimilarityExp_ITcVnColorModel_GUID_6B2F26B1_A1EF_DDE1_974B_94078C6588A7'}
	(* Computes the similarity to a reference color model for each pixel in the source image. (expert function) *)
	FUNCTION F_VN_ReferenceColorSimilarityExp_ITcVnColorModel : HRESULT
	VAR_INPUT
		ipSrcImage	:	ITcVnImage;	(* RGB source image (USINT, 3 channels) *)
		ipDestImage	:	REFERENCE TO ITcVnImage;	(* Returns the similarity to ipColorModel for each pixel in ipSrcImage (USINT, 1 channel. An appropriate destination image will be created if required.) *)
		ipColorModel	:	ITcVnColorModel;	(* Color model *)
		fVariance	:	REAL;	(* Allowed color variance (0.1 - 0.3 might be a good start to try) *)
		fLuminanceWeight	:	REAL;	(* Weight the impact of the luminance ([0..1], e.g. set to 0 to be more resistant to unequal illumination, but might be required to differentiate between some colors. Ignored if ipColorModel is of type RGB.) *)
		hrPrev	:	HRESULT;	(* HRESULT indicating the result of previous operations (If SUCCEEDED(hrPrev) equals false, no operation is executed.) *)
	END_VAR

END_FUNCTION

// Functions/Image Color and Contrast Processing/F_VN_ReferenceColorSimilarity_ITcVnMlModel

	{attribute 'TcIecLibraryType'}
	{attribute 'external_name' := 'F_VN_ReferenceColorSimilarity_ITcVnMlModel_GUID_3F5E6DA4_6A82_D364_8A94_AC91241AFAC7'}
	(* Computes the similarity to a reference color model for each pixel in the source image. *)
	FUNCTION F_VN_ReferenceColorSimilarity_ITcVnMlModel : HRESULT
	VAR_INPUT
		ipSrcImage	:	ITcVnImage;	(* RGB source image (USINT, 3 channels) *)
		ipDestImage	:	REFERENCE TO ITcVnImage;	(* Returns the similarity to ipColorModel for each pixel in ipSrcImage (USINT, 1 channel. An appropriate destination image will be created if required.) *)
		ipColorModel	:	ITcVnMlModel;	(* Color model *)
		hrPrev	:	HRESULT;	(* HRESULT indicating the result of previous operations (If SUCCEEDED(hrPrev) equals false, no operation is executed.) *)
	END_VAR

END_FUNCTION

// Functions/Image Color and Contrast Processing/F_VN_ReferenceColorSimilarityExp_ITcVnMlModel

	{attribute 'TcIecLibraryType'}
	{attribute 'external_name' := 'F_VN_ReferenceColorSimilarityExp_ITcVnMlModel_GUID_1D821506_6C8C_D6F1_BAFD_7E38D4F47482'}
	(* Computes the similarity to a reference color model for each pixel in the source image. (expert function) *)
	FUNCTION F_VN_ReferenceColorSimilarityExp_ITcVnMlModel : HRESULT
	VAR_INPUT
		ipSrcImage	:	ITcVnImage;	(* RGB source image (USINT, 3 channels) *)
		ipDestImage	:	REFERENCE TO ITcVnImage;	(* Returns the similarity to ipColorModel for each pixel in ipSrcImage (USINT, 1 channel. An appropriate destination image will be created if required.) *)
		ipColorModel	:	ITcVnMlModel;	(* Color model *)
		fVariance	:	REAL;	(* Allowed color variance (0.1 - 0.3 might be a good start to try) *)
		fLuminanceWeight	:	REAL;	(* Weight the impact of the luminance ([0..1], e.g. set to 0 to be more resistant to unequal illumination, but might be required to differentiate between some colors. Ignored if ipColorModel is of type RGB.) *)
		hrPrev	:	HRESULT;	(* HRESULT indicating the result of previous operations (If SUCCEEDED(hrPrev) equals false, no operation is executed.) *)
	END_VAR

END_FUNCTION

// Functions/Image Color and Contrast Processing/F_VN_ReferenceColorSimilarity_TcVnVector3_LREAL

	{attribute 'TcIecLibraryType'}
	{attribute 'external_name' := 'F_VN_ReferenceColorSimilarity_TcVnVector3_LREAL_GUID_BFD3E779_1912_D5A2_8237_BEB4F8E75CFC'}
	(* Computes the similarity to a reference color for each pixel in the source image. *)
	FUNCTION F_VN_ReferenceColorSimilarity_TcVnVector3_LREAL : HRESULT
	VAR_INPUT
		ipSrcImage	:	ITcVnImage;	(* RGB source image (USINT, 3 channels) *)
		ipDestImage	:	REFERENCE TO ITcVnImage;	(* Returns the similarity to aRefColor for each pixel in ipSrcImage (USINT, 1 channel. An appropriate destination image will be created if required.) *)
	END_VAR
	VAR_IN_OUT
		aRefColor	:	TcVnVector3_LREAL;	(* Reference color (RGB, [0..255]) *)
	END_VAR
	VAR_INPUT
		hrPrev	:	HRESULT;	(* HRESULT indicating the result of previous operations (If SUCCEEDED(hrPrev) equals false, no operation is executed.) *)
	END_VAR

END_FUNCTION

// Functions/Image Color and Contrast Processing/F_VN_ReferenceColorSimilarityExp_TcVnVector3_LREAL

	{attribute 'TcIecLibraryType'}
	{attribute 'external_name' := 'F_VN_ReferenceColorSimilarityExp_TcVnVector3_LREAL_GUID_9658CC7C_3AF4_DF77_B6EF_EDA71186C4E8'}
	(* Computes the similarity to a reference color for each pixel in the source image. (expert function) *)
	FUNCTION F_VN_ReferenceColorSimilarityExp_TcVnVector3_LREAL : HRESULT
	VAR_INPUT
		ipSrcImage	:	ITcVnImage;	(* RGB source image (USINT, 3 channels) *)
		ipDestImage	:	REFERENCE TO ITcVnImage;	(* Returns the similarity to aRefColor for each pixel in ipSrcImage (USINT, 1 channel. An appropriate destination image will be created if required.) *)
	END_VAR
	VAR_IN_OUT
		aRefColor	:	TcVnVector3_LREAL;	(* Reference color (RGB, [0..255]) *)
	END_VAR
	VAR_INPUT
		fVariance	:	REAL;	(* Allowed color variance (0.1 - 0.3 might be a good start to try) *)
		fLuminanceWeight	:	REAL;	(* Weight the impact of the luminance ([0..1], e.g. set to 0 to be more resistant to unequal illumination, but might be required to differentiate between some colors) *)
		hrPrev	:	HRESULT;	(* HRESULT indicating the result of previous operations (If SUCCEEDED(hrPrev) equals false, no operation is executed.) *)
	END_VAR

END_FUNCTION

// Functions/Image Color and Contrast Processing/F_VN_TrainImageColor

	{attribute 'TcIecLibraryType'}
	{attribute 'external_name' := 'F_VN_TrainImageColor_GUID_47AABA92_1F12_D53F_B661_65549351224C'}
	(* Create a new color model, describing the image color. *)
	FUNCTION F_VN_TrainImageColor : HRESULT
	VAR_INPUT
		ipSrcImage	:	ITcVnImage;	(* Source image (3 channels (RGB) of type USINT) *)
		ipColorModel	:	REFERENCE TO ITcVnColorModel;	(* Returns the color model *)
		nDifferentColors	:	UDINT;	(* Number of different colors to distinguish *)
		hrPrev	:	HRESULT;	(* HRESULT indicating the result of previous operations (If SUCCEEDED(hrPrev) equals false, no operation is executed.) *)
	END_VAR

END_FUNCTION

// Functions/Image Color and Contrast Processing/F_VN_TrainImageColorExp

	{attribute 'TcIecLibraryType'}
	{attribute 'external_name' := 'F_VN_TrainImageColorExp_GUID_247F393B_84B1_D24D_917F_39124AF40BB5'}
	(* Create a new color model, describing the image color. (expert function) *)
	FUNCTION F_VN_TrainImageColorExp : HRESULT
	VAR_INPUT
		ipSrcImage	:	ITcVnImage;	(* Source image (3 channels (RGB) of type USINT) *)
		ipColorModel	:	REFERENCE TO ITcVnColorModel;	(* Returns the color model *)
		nDifferentColors	:	UDINT;	(* Number of different colors to distinguish *)
		eMethod	:	ETcVnColorTrainingMethod;	(* Color training method *)
		ipMask	:	ITcVnImage;	(* Optional image mask (1 channel of type USINT, set to 0 if not required) *)
		nSkipPixels	:	UDINT;	(* Number of pixels to skip between each evaluated color sample (to achieve a better performance). 0 takes every pixel into account and tends to be more accurate. *)
		hrPrev	:	HRESULT;	(* HRESULT indicating the result of previous operations (If SUCCEEDED(hrPrev) equals false, no operation is executed.) *)
	END_VAR

END_FUNCTION

// Functions/Image Color and Contrast Processing/F_VN_TrainImageColorExp2

	{attribute 'TcIecLibraryType'}
	{attribute 'external_name' := 'F_VN_TrainImageColorExp2_GUID_414E7CC2_8C57_DAEF_8308_4458F2756EE3'}
	(* Create a new color model, describing the image color. (expert function) *)
	FUNCTION F_VN_TrainImageColorExp2 : HRESULT
	VAR_INPUT
		ipSrcImage	:	ITcVnImage;	(* Source image (3 channels (RGB) of type USINT) *)
		ipColorModel	:	REFERENCE TO ITcVnColorModel;	(* Returns the color model *)
		nDifferentColors	:	UDINT;	(* Maximum number of different colors to distinguish (if LBG is used as a clustering algorithm, the result might have less different colors, depending on nMaxClusterRadius) *)
		eMethod	:	ETcVnColorTrainingMethod;	(* Color training method *)
		ipMask	:	ITcVnImage;	(* Optional image mask (1 channel of type USINT, set to 0 if not required) *)
		nSkipPixels	:	UDINT;	(* Number of pixels to skip between each evaluated color sample (to achieve a better performance). 0 takes every pixel into account and tends to be more accurate. *)
		eClusteringAlgorithm	:	ETcVnClusteringAlgorithm;	(* Clustering algorithm *)
		nMaxClusterRadius	:	DINT;	(* Only used for the LBG clustering algorithm. Maximum allowed radius (> 0) of a single cluster, i.e. clusters with a higher radius will be split into smaller ones, until a global number of nDifferentColors is reached. *)
		bSingleSplitSteps	:	BOOL;	(* Only used for the LBG clustering algorithm. If true, the global optimization is always run after a single cluster has been split. If false, several clusters are split within the same step before applying the global optimization. Applying the global optimization less often is faster, but can lead to less optimal results, especially having 2 nearby clusters that could be represented by 1) *)
		hrPrev	:	HRESULT;	(* HRESULT indicating the result of previous operations (If SUCCEEDED(hrPrev) equals false, no operation is executed.) *)
	END_VAR

END_FUNCTION

// Functions/Image Color and Contrast Processing/F_VN_TrainImageColor_ITcVnMlModel

	{attribute 'TcIecLibraryType'}
	{attribute 'external_name' := 'F_VN_TrainImageColor_ITcVnMlModel_GUID_0CA9BA92_9C11_D2B5_844B_2669F7129C4B'}
	(* Create a new color model, describing the image color. *)
	FUNCTION F_VN_TrainImageColor_ITcVnMlModel : HRESULT
	VAR_INPUT
		ipSrcImage	:	ITcVnImage;	(* Source image (3 channels (RGB) of type USINT) *)
		ipColorModel	:	REFERENCE TO ITcVnMlModel;	(* Returns the color model *)
		nDifferentColors	:	UDINT;	(* Number of different colors to distinguish *)
		hrPrev	:	HRESULT;	(* HRESULT indicating the result of previous operations (If SUCCEEDED(hrPrev) equals false, no operation is executed.) *)
	END_VAR

END_FUNCTION

// Functions/Image Color and Contrast Processing/F_VN_TrainImageColorExp_ITcVnMlModel

	{attribute 'TcIecLibraryType'}
	{attribute 'external_name' := 'F_VN_TrainImageColorExp_ITcVnMlModel_GUID_AF47CE9C_D358_D021_BB58_8CAA556D47B5'}
	(* Create a new color model, describing the image color. (expert function) *)
	FUNCTION F_VN_TrainImageColorExp_ITcVnMlModel : HRESULT
	VAR_INPUT
		ipSrcImage	:	ITcVnImage;	(* Source image (3 channels (RGB) of type USINT) *)
		ipColorModel	:	REFERENCE TO ITcVnMlModel;	(* Returns the color model *)
		nDifferentColors	:	UDINT;	(* Number of different colors to distinguish *)
		eMethod	:	ETcVnColorTrainingMethod;	(* Color training method *)
		ipMask	:	ITcVnImage;	(* Optional image mask (1 channel of type USINT, set to 0 if not required) *)
		nSkipPixels	:	UDINT;	(* Number of pixels to skip between each evaluated color sample (to achieve a better performance). 0 takes every pixel into account and tends to be more accurate. *)
		hrPrev	:	HRESULT;	(* HRESULT indicating the result of previous operations (If SUCCEEDED(hrPrev) equals false, no operation is executed.) *)
	END_VAR

END_FUNCTION

// Functions/Image Color and Contrast Processing/F_VN_TrainImageColorExp2_ITcVnMlModel

	{attribute 'TcIecLibraryType'}
	{attribute 'external_name' := 'F_VN_TrainImageColorExp2_ITcVnMlModel_GUID_177D7547_7FAC_D8F4_8885_BDC290EBE602'}
	(* Create a new color model, describing the image color. (expert function) *)
	FUNCTION F_VN_TrainImageColorExp2_ITcVnMlModel : HRESULT
	VAR_INPUT
		ipSrcImage	:	ITcVnImage;	(* Source image (3 channels (RGB) of type USINT) *)
		ipColorModel	:	REFERENCE TO ITcVnMlModel;	(* Returns the color model *)
		nDifferentColors	:	UDINT;	(* Maximum number of different colors to distinguish (if LBG is used as a clustering algorithm, the result might have less different colors, depending on nMaxClusterRadius) *)
		eMethod	:	ETcVnColorTrainingMethod;	(* Color training method *)
		ipMask	:	ITcVnImage;	(* Optional image mask (1 channel of type USINT, set to 0 if not required) *)
		nSkipPixels	:	UDINT;	(* Number of pixels to skip between each evaluated color sample (to achieve a better performance). 0 takes every pixel into account and tends to be more accurate. *)
		eClusteringAlgorithm	:	ETcVnClusteringAlgorithm;	(* Clustering algorithm *)
		nMaxClusterRadius	:	DINT;	(* Only used for the LBG clustering algorithm. Maximum allowed radius (> 0) of a single cluster, i.e. clusters with a higher radius will be split into smaller ones, until a global number of nDifferentColors is reached. *)
		bSingleSplitSteps	:	BOOL;	(* Only used for the LBG clustering algorithm. If true, the global optimization is always run after a single cluster has been split. If false, several clusters are split within the same step before applying the global optimization. Applying the global optimization less often is faster, but can lead to less optimal results, especially having 2 nearby clusters that could be represented by 1) *)
		hrPrev	:	HRESULT;	(* HRESULT indicating the result of previous operations (If SUCCEEDED(hrPrev) equals false, no operation is executed.) *)
	END_VAR

END_FUNCTION

// Functions/Image Color and Contrast Processing/F_VN_WhiteBalance

	{attribute 'TcIecLibraryType'}
	{attribute 'external_name' := 'F_VN_WhiteBalance_GUID_DF2C9DCB_DA3C_DA85_A401_BE771738A9BD'}
	(* Calculates the white balance ratios for a RGB image. Uses the green channel as a reference and computes the relative ratios for the red and blue channels. Requires a non-reflecting, not overexposed white colored object (e.g. a sheet of paper) in at least 100 pixels of the image to provide reasonable results. The resulting ratios can then be set on the camera (multiply with existing ratios), or applied in the PLC via MultiplyImageWithVector. *)
	FUNCTION F_VN_WhiteBalance : HRESULT
	VAR_INPUT
		ipSrcImage	:	ITcVnImage;	(* Source image (3 channels (RGB), USINT or UINT) *)
		ipDestImage	:	REFERENCE TO ITcVnImage;	(* Destination image with white balance applied (optional, set to 0 if not required. An appropriate image will be created if required.) *)
		fRatioRed	:	REFERENCE TO REAL;	(* Returns the ratio for the red channel *)
		fRatioBlue	:	REFERENCE TO REAL;	(* Returns the ratio for the blue channel *)
		nMaxValue	:	UDINT;	(* Specify the maximum pixel value that would be achieved by overexposure (usually 255 for 8 bit or 4095 for 12 bit data) *)
		hrPrev	:	HRESULT;	(* HRESULT indicating the result of previous operations (If SUCCEEDED(hrPrev) equals false, no operation is executed.) *)
	END_VAR

END_FUNCTION

// Functions/Contour Analysis/F_VN_ApproximatePolygon

	{attribute 'TcIecLibraryType'}
	{attribute 'external_name' := 'F_VN_ApproximatePolygon_GUID_E359F294_E792_D763_8C24_88CCE9F5F94D'}
	(* Approximate a contour to a simplified polygon (using the Douglas-Peucker algorithm). *)
	FUNCTION F_VN_ApproximatePolygon : HRESULT
	VAR_INPUT
		ipSrcContour	:	ITcVnContainer;	(* Single contour (ContainerType_Vector_TcVnPoint2_DINT or ContainerType_Vector_TcVnPoint2_REAL; The elements of this container are the points of the contour.) *)
		ipDestContour	:	REFERENCE TO ITcVnContainer;	(* Returns a container which is filled with the approximated polygon points (same type ID as ipSrcContour; Non-zero interface pointers are reused.) *)
		fMaxDist	:	LREAL;	(* Maximum distance between the original contour and its approximation *)
		bClosed	:	BOOL;	(* Specify, if the contour is closed (first and last points connected) or not *)
		hrPrev	:	HRESULT;	(* HRESULT indicating the result of previous operations (If SUCCEEDED(hrPrev) equals false, no operation is executed.) *)
	END_VAR

END_FUNCTION

// Functions/Contour Analysis/F_VN_CheckIfPointIsInsideContour

	{attribute 'TcIecLibraryType'}
	{attribute 'external_name' := 'F_VN_CheckIfPointIsInsideContour_GUID_265CF2CF_E0E7_D908_9039_642769A1F3FF'}
	(* Checks if a point is inside a contour (and optionally return the distance to it). *)
	FUNCTION F_VN_CheckIfPointIsInsideContour : HRESULT
	VAR_INPUT
		ipContour	:	ITcVnContainer;	(* Single contour (ContainerType_Vector_TcVnPoint2_DINT or ContainerType_Vector_TcVnPoint2_REAL) *)
	END_VAR
	VAR_IN_OUT
		aPoint	:	TcVnPoint2_REAL;	(* Point position to check *)
		fDist	:	LREAL;	(* Returns the result (> 0: the point is inside the contour; 0: the point is on the contour; < 0: the point is outside the contour) *)
	END_VAR
	VAR_INPUT
		bMeasureDistance	:	BOOL;	(* If true, fDist returns the distance to the nearest contour edge. Otherwise, fDist only returns -1, 0 or +1 (recommended to set to false if the distance is not required, as this is faster). *)
		hrPrev	:	HRESULT;	(* HRESULT indicating the result of previous operations (If SUCCEEDED(hrPrev) equals false, no operation is executed.) *)
	END_VAR

END_FUNCTION

// Functions/Contour Analysis/F_VN_ContourArea

	{attribute 'TcIecLibraryType'}
	{attribute 'external_name' := 'F_VN_ContourArea_GUID_F796A806_656A_D006_BAFC_3EBBB8E34C61'}
	(* Estimate the contour area using Green's formula. *)
	FUNCTION F_VN_ContourArea : HRESULT
	VAR_INPUT
		ipContour	:	ITcVnContainer;	(* Single contour (ContainerType_Vector_TcVnPoint2_DINT or ContainerType_Vector_TcVnPoint2_REAL; The elements of this container are the points of the contour.) *)
	END_VAR
	VAR_IN_OUT
		fArea	:	LREAL;	(* Returns the estimated contour area (The actual contour area may differ depending on the shape of the contour.) *)
	END_VAR
	VAR_INPUT
		hrPrev	:	HRESULT;	(* HRESULT indicating the result of previous operations (If SUCCEEDED(hrPrev) equals false, no operation is executed.) *)
	END_VAR

END_FUNCTION

// Functions/Contour Analysis/F_VN_ContourCenterOfMass

	{attribute 'TcIecLibraryType'}
	{attribute 'external_name' := 'F_VN_ContourCenterOfMass_GUID_4BF2F257_C13F_D4F9_ADB5_C85825230B5C'}
	(* Computes the center of mass of a contour. *)
	FUNCTION F_VN_ContourCenterOfMass : HRESULT
	VAR_INPUT
		ipContour	:	ITcVnContainer;	(* Single contour (ContainerType_Vector_TcVnPoint2_DINT or ContainerType_Vector_TcVnPoint2_REAL; The elements of this container are the points of the contour.) *)
	END_VAR
	VAR_IN_OUT
		aCenterOfMass	:	TcVnPoint2_LREAL;	(* Returns the center of mass of the contour *)
	END_VAR
	VAR_INPUT
		hrPrev	:	HRESULT;	(* HRESULT indicating the result of previous operations (If SUCCEEDED(hrPrev) equals false, no operation is executed.) *)
	END_VAR

END_FUNCTION

// Functions/Contour Analysis/F_VN_ContourCircularity

	{attribute 'TcIecLibraryType'}
	{attribute 'external_name' := 'F_VN_ContourCircularity_GUID_B1194450_C4B8_DC33_A36D_CB186948697A'}
	(* Computes the circularity of a contour (1.0: ideal circle, 0.0: straight line). *)
	FUNCTION F_VN_ContourCircularity : HRESULT
	VAR_INPUT
		ipContour	:	ITcVnContainer;	(* Single contour (ContainerType_Vector_TcVnPoint2_DINT or ContainerType_Vector_TcVnPoint2_REAL; The elements of this container are the points of the contour.) *)
	END_VAR
	VAR_IN_OUT
		fCircularity	:	LREAL;	(* Returns the circularity of the contour [0..1] *)
	END_VAR
	VAR_INPUT
		hrPrev	:	HRESULT;	(* HRESULT indicating the result of previous operations (If SUCCEEDED(hrPrev) equals false, no operation is executed.) *)
	END_VAR

END_FUNCTION

// Functions/Contour Analysis/F_VN_ContourCircularityExp

	{attribute 'TcIecLibraryType'}
	{attribute 'external_name' := 'F_VN_ContourCircularityExp_GUID_C1C0619D_6DA9_D45C_8A0A_11FED2AA91B4'}
	(* Computes the circularity of a contour (1.0: ideal circle, 0.0: straight line). (expert function) *)
	FUNCTION F_VN_ContourCircularityExp : HRESULT
	VAR_INPUT
		ipContour	:	ITcVnContainer;	(* Single contour (ContainerType_Vector_TcVnPoint2_DINT or ContainerType_Vector_TcVnPoint2_REAL; The elements of this container are the points of the contour.) *)
	END_VAR
	VAR_IN_OUT
		fCircularity	:	LREAL;	(* Returns the circularity of the contour [0..1] *)
	END_VAR
	VAR_INPUT
		eMethod	:	ETcVnCircularityCalculationMethod;	(* Method used for computing the circularity *)
		hrPrev	:	HRESULT;	(* HRESULT indicating the result of previous operations (If SUCCEEDED(hrPrev) equals false, no operation is executed.) *)
	END_VAR

END_FUNCTION

// Functions/Contour Analysis/F_VN_ContourConvexity

	{attribute 'TcIecLibraryType'}
	{attribute 'external_name' := 'F_VN_ContourConvexity_GUID_5F77DE11_E331_DBB0_85CB_CD6F494EE931'}
	(* Computes the convexity of a contour as the ratio between the contour's area and the area of the convex hull (1.0: convex shapes (i.e. rectangle, circle, ..., etc.), 0.0: zero area (i.e. a line or an empty contour)). *)
	FUNCTION F_VN_ContourConvexity : HRESULT
	VAR_INPUT
		ipContour	:	ITcVnContainer;	(* Single contour (ContainerType_Vector_TcVnPoint2_DINT or ContainerType_Vector_TcVnPoint2_REAL; The elements of this container are the points of the contour.) *)
	END_VAR
	VAR_IN_OUT
		fConvexity	:	LREAL;	(* Returns the convexity of the contour [0..1] *)
	END_VAR
	VAR_INPUT
		hrPrev	:	HRESULT;	(* HRESULT indicating the result of previous operations (If SUCCEEDED(hrPrev) equals false, no operation is executed.) *)
	END_VAR

END_FUNCTION

// Functions/Contour Analysis/F_VN_ContourEccentricity

	{attribute 'TcIecLibraryType'}
	{attribute 'external_name' := 'F_VN_ContourEccentricity_GUID_D0ABD9BF_3136_D572_8F41_62FCBBB2ACB0'}
	(* Computes the eccentricity of a contour (0.0: circular, 1.0: linear). *)
	FUNCTION F_VN_ContourEccentricity : HRESULT
	VAR_INPUT
		ipContour	:	ITcVnContainer;	(* Single contour (ContainerType_Vector_TcVnPoint2_DINT or ContainerType_Vector_TcVnPoint2_REAL; The elements of this container are the points of the contour.) *)
	END_VAR
	VAR_IN_OUT
		fEccentricity	:	LREAL;	(* Returns the eccentricity of the contour [0..1] *)
	END_VAR
	VAR_INPUT
		hrPrev	:	HRESULT;	(* HRESULT indicating the result of previous operations (If SUCCEEDED(hrPrev) equals false, no operation is executed.) *)
	END_VAR

END_FUNCTION

// Functions/Contour Analysis/F_VN_ContourElongation

	{attribute 'TcIecLibraryType'}
	{attribute 'external_name' := 'F_VN_ContourElongation_GUID_7DAC4A1C_ED46_D391_895A_55774677184C'}
	(* Computes the elongation factor of a contour. *)
	FUNCTION F_VN_ContourElongation : HRESULT
	VAR_INPUT
		ipContour	:	ITcVnContainer;	(* Single contour (ContainerType_Vector_TcVnPoint2_DINT or ContainerType_Vector_TcVnPoint2_REAL; The elements of this container are the points of the contour.) *)
	END_VAR
	VAR_IN_OUT
		fElongation	:	LREAL;	(* Returns the elongation of the contour *)
	END_VAR
	VAR_INPUT
		hrPrev	:	HRESULT;	(* HRESULT indicating the result of previous operations (If SUCCEEDED(hrPrev) equals false, no operation is executed.) *)
	END_VAR

END_FUNCTION

// Functions/Contour Analysis/F_VN_ContourExtremePoint

	{attribute 'TcIecLibraryType'}
	{attribute 'external_name' := 'F_VN_ContourExtremePoint_GUID_A00FCB73_D74E_DA35_8270_799FB71CBE9B'}
	(* Finds the contour extreme point. *)
	FUNCTION F_VN_ContourExtremePoint : HRESULT
	VAR_INPUT
		ipContour	:	ITcVnContainer;	(* Source container with 2D points (TcVnPoint2_DINT or TcVnPoint2_REAL or TcVnPoint2_LREAL) *)
		eDirection	:	ETcVnExtremePointDirection;	(* Selects the search direction for the extreme point *)
	END_VAR
	VAR_IN_OUT
		aExtremePoint	:	TcVnPoint2_LREAL;	(* Returns the extreme point of the contour, according to eDirection *)
	END_VAR
	VAR_INPUT
		hrPrev	:	HRESULT;	(* HRESULT indicating the result of previous operations (If SUCCEEDED(hrPrev) equals false, no operation is executed.) *)
	END_VAR

END_FUNCTION

// Functions/Contour Analysis/F_VN_ContourInertiaRatio

	{attribute 'TcIecLibraryType'}
	{attribute 'external_name' := 'F_VN_ContourInertiaRatio_GUID_B8B4B1BE_DBDA_D5AD_98D5_25EB5CEF4573'}
	(* Computes the inertia ratio of a contour which reflects how a contour/shape is elongated (i.e. circle: 1.0, line: 0.0). *)
	FUNCTION F_VN_ContourInertiaRatio : HRESULT
	VAR_INPUT
		ipContour	:	ITcVnContainer;	(* Single contour (ContainerType_Vector_TcVnPoint2_DINT or ContainerType_Vector_TcVnPoint2_REAL; The elements of this container are the points of the contour.) *)
	END_VAR
	VAR_IN_OUT
		fInertiaRatio	:	LREAL;	(* Returns the inertia raio of the contour [0..1] *)
	END_VAR
	VAR_INPUT
		hrPrev	:	HRESULT;	(* HRESULT indicating the result of previous operations (If SUCCEEDED(hrPrev) equals false, no operation is executed.) *)
	END_VAR

END_FUNCTION

// Functions/Contour Analysis/F_VN_ContourMoments

	{attribute 'TcIecLibraryType'}
	{attribute 'external_name' := 'F_VN_ContourMoments_GUID_D5B03DA4_EDDB_DDD6_8E54_659C74B852BC'}
	(* Computes the spatial moments, the central moments, and the central normalized moments of a contour up to the third order. *)
	FUNCTION F_VN_ContourMoments : HRESULT
	VAR_INPUT
		ipContour	:	ITcVnContainer;	(* Single contour (ContainerType_Vector_TcVnPoint2_DINT or ContainerType_Vector_TcVnPoint2_REAL; The elements of this container are the points of the contour.) *)
	END_VAR
	VAR_IN_OUT
		stMoments	:	TcVnMoments;	(* Returns a struct containing the moments *)
	END_VAR
	VAR_INPUT
		hrPrev	:	HRESULT;	(* HRESULT indicating the result of previous operations (If SUCCEEDED(hrPrev) equals false, no operation is executed.) *)
	END_VAR

END_FUNCTION

// Functions/Contour Analysis/F_VN_ContourOrientation

	{attribute 'TcIecLibraryType'}
	{attribute 'external_name' := 'F_VN_ContourOrientation_GUID_A1B75AC4_8716_DFB6_B97B_2078D35876CC'}
	(* Calculate the orientation of a contour or a set of points. *)
	FUNCTION F_VN_ContourOrientation : HRESULT
	VAR_INPUT
		ipContour	:	ITcVnContainer;	(* Source point set (ContainerType_Vector_TcVnPoint2_DINT, ContainerType_Vector_TcVnPoint2_REAL, or ContainerType_Vector_TcVnPoint2_LREAL. The elements of this container are the individual points.) *)
	END_VAR
	VAR_IN_OUT
		stOrientation	:	TcVnRotatedRectangle;	(* Resulting rotated rectangle, containig center of mass, lenghts of axes, and rotation angle of the contour in clockwise direction. *)
	END_VAR
	VAR_INPUT
		hrPrev	:	HRESULT;	(* HRESULT indicating the result of previous operations (If SUCCEEDED(hrPrev) equals false, no operation is executed.) *)
	END_VAR

END_FUNCTION

// Functions/Contour Analysis/F_VN_ContourOrientationExp

	{attribute 'TcIecLibraryType'}
	{attribute 'external_name' := 'F_VN_ContourOrientationExp_GUID_7597E595_47A9_DD26_97E4_DE583EE94374'}
	(* Calculate the orientation of a contour or a set of points. (expert function) *)
	FUNCTION F_VN_ContourOrientationExp : HRESULT
	VAR_INPUT
		ipContour	:	ITcVnContainer;	(* Source point set (ContainerType_Vector_TcVnPoint2_DINT, ContainerType_Vector_TcVnPoint2_REAL, or ContainerType_Vector_TcVnPoint2_LREAL. The elements of this container are the individual points.) *)
	END_VAR
	VAR_IN_OUT
		stOrientation	:	TcVnRotatedRectangle;	(* Resulting rotated rectangle, containig center of mass, lenghts of axes, and rotation angle of the contour in clockwise direction. *)
	END_VAR
	VAR_INPUT
		eMethod	:	ETcVnOrientationMethod;	(* Method for calculating the orientation.  *)
		hrPrev	:	HRESULT;	(* HRESULT indicating the result of previous operations (If SUCCEEDED(hrPrev) equals false, no operation is executed.) *)
	END_VAR

END_FUNCTION

// Functions/Contour Analysis/F_VN_ContourPerimeter

	{attribute 'TcIecLibraryType'}
	{attribute 'external_name' := 'F_VN_ContourPerimeter_GUID_E52B35F1_6558_D91B_8AB3_A4E51F5AF5DB'}
	(* Computes the perimeter of a contour (curve length if the contour is not closed). *)
	FUNCTION F_VN_ContourPerimeter : HRESULT
	VAR_INPUT
		ipContour	:	ITcVnContainer;	(* Single contour (ContainerType_Vector_TcVnPoint2_DINT or ContainerType_Vector_TcVnPoint2_REAL; The elements of this container are the points of the contour.) *)
	END_VAR
	VAR_IN_OUT
		fPerimeter	:	LREAL;	(* Returns the perimeter of the contour *)
	END_VAR
	VAR_INPUT
		bClosed	:	BOOL;	(* Specifys, if the contour is closed (first and last points connected) or not *)
		hrPrev	:	HRESULT;	(* HRESULT indicating the result of previous operations (If SUCCEEDED(hrPrev) equals false, no operation is executed.) *)
	END_VAR

END_FUNCTION

// Functions/Contour Analysis/F_VN_ContourRoundness

	{attribute 'TcIecLibraryType'}
	{attribute 'external_name' := 'F_VN_ContourRoundness_GUID_26580415_F70F_D0A3_949A_2D62E3787DAC'}
	(* Computes the roundness of a contour (perimeter^2 / area). *)
	FUNCTION F_VN_ContourRoundness : HRESULT
	VAR_INPUT
		ipContour	:	ITcVnContainer;	(* Single contour (ContainerType_Vector_TcVnPoint2_DINT or ContainerType_Vector_TcVnPoint2_REAL; The elements of this container are the points of the contour.) *)
	END_VAR
	VAR_IN_OUT
		fRoundness	:	LREAL;	(* Returns the roundness of the contour *)
	END_VAR
	VAR_INPUT
		hrPrev	:	HRESULT;	(* HRESULT indicating the result of previous operations (If SUCCEEDED(hrPrev) equals false, no operation is executed.) *)
	END_VAR

END_FUNCTION

// Functions/Contour Analysis/F_VN_ConvexHullPoints

	{attribute 'TcIecLibraryType'}
	{attribute 'external_name' := 'F_VN_ConvexHullPoints_GUID_7CFF123C_4058_D05D_8E26_A90FC6F074B8'}
	(* Determines the convex hull of a point set. *)
	FUNCTION F_VN_ConvexHullPoints : HRESULT
	VAR_INPUT
		ipPointSet	:	ITcVnContainer;	(* Source point set (ContainerType_Vector_TcVnPoint2_DINT or ContainerType_Vector_TcVnPoint2_REAL; The elements of this container are the individual points.) *)
		ipConvexHull	:	REFERENCE TO ITcVnContainer;	(* Returns a container which is filled with the sorted convex hull points (same type ID as ipPointSet; Non-zero interface pointers are reused.) *)
		hrPrev	:	HRESULT;	(* HRESULT indicating the result of previous operations (If SUCCEEDED(hrPrev) equals false, no operation is executed.) *)
	END_VAR

END_FUNCTION

// Functions/Contour Analysis/F_VN_ConvexHullPointsExp

	{attribute 'TcIecLibraryType'}
	{attribute 'external_name' := 'F_VN_ConvexHullPointsExp_GUID_314F1D5E_1C2E_D708_B1BC_2C0110A6BD51'}
	(* Determines the convex hull of a point set. (expert function) *)
	FUNCTION F_VN_ConvexHullPointsExp : HRESULT
	VAR_INPUT
		ipPointSet	:	ITcVnContainer;	(* Source point set (ContainerType_Vector_TcVnPoint2_DINT or ContainerType_Vector_TcVnPoint2_REAL; The elements of this container are the individual points.) *)
		ipConvexHull	:	REFERENCE TO ITcVnContainer;	(* Returns a container which is filled with the sorted convex hull points (same type ID as ipPointSet; Non-zero interface pointers are reused.) *)
		bClockwise	:	BOOL;	(* Selects the sorting direction of the hull points, assuming cartesian coordinates. *)
		hrPrev	:	HRESULT;	(* HRESULT indicating the result of previous operations (If SUCCEEDED(hrPrev) equals false, no operation is executed.) *)
	END_VAR

END_FUNCTION

// Functions/Contour Analysis/F_VN_ConvexityDefects

	{attribute 'TcIecLibraryType'}
	{attribute 'external_name' := 'F_VN_ConvexityDefects_GUID_FBED5BEE_F7D8_D648_85E8_63DD4096B732'}
	(* Finds the convexity defects of a point set. *)
	FUNCTION F_VN_ConvexityDefects : HRESULT
	VAR_INPUT
		ipContour	:	ITcVnContainer;	(* Source contour (ContainerType_Vector_TcVnPoint2_DINT; The elements of this container are the individual points.) *)
		ipConvexityDefects	:	REFERENCE TO ITcVnContainer;	(* Returns a container which is filled with the convexity defects (ContainerType_Vector_TcVnVector4_DINT with [startIndex, endIndex, furthestPointIndex, fixedPointDistance (8 fraction bits, i.e. divide by 256 to get the distance in pixels)]; Non-zero interface pointers are reused.) *)
		hrPrev	:	HRESULT;	(* HRESULT indicating the result of previous operations (If SUCCEEDED(hrPrev) equals false, no operation is executed.) *)
	END_VAR

END_FUNCTION

// Functions/Contour Analysis/F_VN_CustomElementWiseContainerOperation_ITcVnContainer

	{attribute 'TcIecLibraryType'}
	{attribute 'external_name' := 'F_VN_CustomElementWiseContainerOperation_ITcVnContainer_GUID_A4262FE6_CA73_D83B_BBD6_765AA2543C91'}
	(* Performs a custom, element wise operation on a set of up to 3 containers. *)
	FUNCTION F_VN_CustomElementWiseContainerOperation_ITcVnContainer : HRESULT
	VAR_INPUT
		ipContainer1	:	ITcVnContainer;	(* Container 1 *)
		ipContainer2	:	ITcVnContainer;	(* Container 2 *)
		ipContainer3	:	ITcVnContainer;	(* Container 3 *)
		ipOperationFB	:	ITcVnCustomContainerOperation_ITcVnContainer;	(* Custom operation on the container elements *)
		hrPrev	:	HRESULT;	(* HRESULT indicating the result of previous operations (If SUCCEEDED(hrPrev) equals false, no operation is executed.) *)
	END_VAR

END_FUNCTION

// Interfaces/Containers/Function Blocks/ITcVnCustomContainerOperation_ITcVnContainer

	(* Offers an interface for custom, elementwise container operations (for containers of containers) with up to 3 different containers. *)
	{attribute 'c++_compatible'}
	INTERFACE ITcVnCustomContainerOperation_ITcVnContainer


(* Executes the custom operation on the container elements. *)
	{attribute 'c++_compatible'}
	{attribute 'minimal_input_size' := '4'}
	{attribute 'pack_mode' := '4'}
	METHOD Execute : HRESULT
	VAR_INPUT
		ipElement1 : ITcVnContainer;
		ipElement2 : ITcVnContainer;
		ipElement3 : ITcVnContainer;
	END_VAR
END_METHOD

END_INTERFACE

// Functions/Contour Analysis/F_VN_CustomElementWiseContainerOperation_ITcVnForwardIterator

	{attribute 'TcIecLibraryType'}
	{attribute 'external_name' := 'F_VN_CustomElementWiseContainerOperation_ITcVnForwardIterator_GUID_8C8C1911_AB87_D83F_AC23_561C5E028828'}
	(* Performs a custom, element wise operation on a set of up to 3 containers. *)
	FUNCTION F_VN_CustomElementWiseContainerOperation_ITcVnForwardIterator : HRESULT
	VAR_INPUT
		ipContainer1	:	ITcVnContainer;	(* Container 1 *)
		ipContainer2	:	ITcVnContainer;	(* Container 2 *)
		ipContainer3	:	ITcVnContainer;	(* Container 3 *)
		ipOperationFB	:	ITcVnCustomContainerOperation_ITcVnForwardIterator;	(* Custom operation on the elements *)
		hrPrev	:	HRESULT;	(* HRESULT indicating the result of previous operations (If SUCCEEDED(hrPrev) equals false, no operation is executed.) *)
	END_VAR

END_FUNCTION

// Interfaces/Containers/Function Blocks/ITcVnCustomContainerOperation_ITcVnForwardIterator

	(* Offers an interface for custom, elementwise container operations with up to 3 different containers. *)
	{attribute 'c++_compatible'}
	INTERFACE ITcVnCustomContainerOperation_ITcVnForwardIterator


(* Executes the custom operation on the container elements. *)
	{attribute 'c++_compatible'}
	{attribute 'minimal_input_size' := '4'}
	{attribute 'pack_mode' := '4'}
	METHOD Execute : HRESULT
	VAR_INPUT
		ipElement1 : ITcVnForwardIterator;
		ipElement2 : ITcVnForwardIterator;
		ipElement3 : ITcVnForwardIterator;
	END_VAR
END_METHOD

END_INTERFACE

// Functions/Contour Analysis/F_VN_EnclosingCircle

	{attribute 'TcIecLibraryType'}
	{attribute 'external_name' := 'F_VN_EnclosingCircle_GUID_033016AC_EBC4_D1A8_BA21_642F01EE5FFD'}
	(* Searchs for a minimum area circle enclosing a set of points. *)
	FUNCTION F_VN_EnclosingCircle : HRESULT
	VAR_INPUT
		ipPointSet	:	ITcVnContainer;	(* Source point set (ContainerType_Vector_TcVnPoint2_DINT or ContainerType_Vector_TcVnPoint2_REAL; The elements of this container are the individual points.) *)
	END_VAR
	VAR_IN_OUT
		aCenter	:	TcVnPoint2_REAL;	(* Returns the center of the circle *)
		fRadius	:	REAL;	(* Returns the radius of the circle *)
	END_VAR
	VAR_INPUT
		hrPrev	:	HRESULT;	(* HRESULT indicating the result of previous operations (If SUCCEEDED(hrPrev) equals false, no operation is executed.) *)
	END_VAR

END_FUNCTION

// Functions/Contour Analysis/F_VN_EnclosingRectangle

	{attribute 'TcIecLibraryType'}
	{attribute 'external_name' := 'F_VN_EnclosingRectangle_GUID_756776DF_4CD3_D5C7_A267_45DDAB2E587D'}
	(* Searches for a minimum area rectangle enclosing a set of points. *)
	FUNCTION F_VN_EnclosingRectangle : HRESULT
	VAR_INPUT
		ipPointSet	:	ITcVnContainer;	(* Source point set (ContainerType_Vector_TcVnPoint2_DINT or ContainerType_Vector_TcVnPoint2_REAL; The elements of this container are the individual points.) *)
	END_VAR
	VAR_IN_OUT
		stRectangle	:	TcVnRotatedRectangle;	(* Returns the determined rectangle *)
	END_VAR
	VAR_INPUT
		hrPrev	:	HRESULT;	(* HRESULT indicating the result of previous operations (If SUCCEEDED(hrPrev) equals false, no operation is executed.) *)
	END_VAR

END_FUNCTION

// Functions/Contour Analysis/F_VN_EnclosingTriangle

	{attribute 'TcIecLibraryType'}
	{attribute 'external_name' := 'F_VN_EnclosingTriangle_GUID_B89BDC81_9039_DBB8_87C8_27545986C187'}
	(* Searches for a minimum area triangle enclosing a set of points. *)
	FUNCTION F_VN_EnclosingTriangle : HRESULT
	VAR_INPUT
		ipPointSet	:	ITcVnContainer;	(* Source point set (ContainerType_Vector_TcVnPoint2_DINT or ContainerType_Vector_TcVnPoint2_REAL; The elements of this container are the individual points.) *)
	END_VAR
	VAR_IN_OUT
		aTriangleVertices	:	TcVnArray3_Point2_REAL;	(* Returns the 3 triangle vertices *)
	END_VAR
	VAR_INPUT
		hrPrev	:	HRESULT;	(* HRESULT indicating the result of previous operations (If SUCCEEDED(hrPrev) equals false, no operation is executed.) *)
	END_VAR
	VAR_OUTPUT
		fArea	:	LREAL;	(* Returns the triangle area *)
	END_VAR

END_FUNCTION

// Functions/Contour Analysis/F_VN_FitEllipse

	{attribute 'TcIecLibraryType'}
	{attribute 'external_name' := 'F_VN_FitEllipse_GUID_BE2FF5CE_1D13_D11A_BB55_CED2371B31C9'}
	(* Fit an ellipse in a point set. *)
	FUNCTION F_VN_FitEllipse : HRESULT
	VAR_INPUT
		ipPointSet	:	ITcVnContainer;	(* Source point set (ContainerType_Vector_TcVnPoint2_DINT or ContainerType_Vector_TcVnPoint2_REAL; At least 5 reasonable points are required! The elements of this container are the individual points.) *)
	END_VAR
	VAR_IN_OUT
		stEllipse	:	TcVnRotatedRectangle;	(* Resulting ellipse, described by a rotated rectangle. *)
	END_VAR
	VAR_INPUT
		hrPrev	:	HRESULT;	(* HRESULT indicating the result of previous operations (If SUCCEEDED(hrPrev) equals false, no operation is executed.) *)
	END_VAR

END_FUNCTION

// Functions/Contour Analysis/F_VN_FitLine

	{attribute 'TcIecLibraryType'}
	{attribute 'external_name' := 'F_VN_FitLine_GUID_9E39439F_2E35_DA2D_9EB3_9586853D906C'}
	(* Fit a line into a point set. *)
	FUNCTION F_VN_FitLine : HRESULT
	VAR_INPUT
		ipPointSet	:	ITcVnContainer;	(* Source point set (ContainerType_Vector_TcVnPoint2_DINT or ContainerType_Vector_TcVnPoint2_REAL; The elements of this container are the individual points.) *)
	END_VAR
	VAR_IN_OUT
		aFitLine	:	TcVnVector4_LREAL;	(* Resulting line. The first and second element describe the x and y component of a vector collinear to the line. The third and fourth element describe the x and y component of a point on the line. *)
	END_VAR
	VAR_INPUT
		hrPrev	:	HRESULT;	(* HRESULT indicating the result of previous operations (If SUCCEEDED(hrPrev) equals false, no operation is executed.) *)
	END_VAR

END_FUNCTION

// Functions/Contour Analysis/F_VN_FitLineExp

	{attribute 'TcIecLibraryType'}
	{attribute 'external_name' := 'F_VN_FitLineExp_GUID_56F24665_0B1E_D18A_A60F_5B9250D02618'}
	(* Fit a line into a point set. (expert function) *)
	FUNCTION F_VN_FitLineExp : HRESULT
	VAR_INPUT
		ipPointSet	:	ITcVnContainer;	(* Source point set (ContainerType_Vector_TcVnPoint2_DINT or ContainerType_Vector_TcVnPoint2_REAL; The elements of this container are the individual points.) *)
	END_VAR
	VAR_IN_OUT
		aFitLine	:	TcVnVector4_LREAL;	(* Resulting line. The first and second element describe the x and y component of a vector collinear to the line. The third and fourth element describe the x and y component of a point on the line. *)
	END_VAR
	VAR_INPUT
		eDistanceType	:	ETcVnDistanceType;	(* Distance computation method (supported: L1, L2, L12, FAIR, WELSCH, HUBER) *)
		fParam	:	LREAL;	(* Numerical parameter (c) for some eDistanceType (should be >= 0). If 0, an optimal value is chosen internally. *)
		fEpsRadius	:	LREAL;	(* Accuracy of the radius (distance of the line from the coordinate origin, should be > 0). A smaller value means higher accuracy. *)
		fEpsAngle	:	LREAL;	(* Accuracy of the angle (should be > 0). A smaller value means higher accuracy. *)
		hrPrev	:	HRESULT;	(* HRESULT indicating the result of previous operations (If SUCCEEDED(hrPrev) equals false, no operation is executed.) *)
	END_VAR

END_FUNCTION

// Functions/Contour Analysis/F_VN_FourierDescriptors

	{attribute 'TcIecLibraryType'}
	{attribute 'external_name' := 'F_VN_FourierDescriptors_GUID_0748C1DA_ACC4_DC64_8D82_AFFAC52907E4'}
	(* Computes the fourier descriptors for a closed contour. *)
	FUNCTION F_VN_FourierDescriptors : HRESULT
	VAR_INPUT
		ipContour	:	ITcVnContainer;	(* Closed contour (ContainerType_Vector_TcVnPoint2_DINT or ContainerType_Vector_TcVnPoint2_REAL or ContainerType_Vector_TcVnPoint2_LREAL. Providing the full contour is strongly recommended, i.e. use TCVN_CAM_NONE for contour detection algorithms.) *)
		ipDescriptors	:	REFERENCE TO ITcVnContainer;	(* Returns the fourier descriptors for ipContour (Re0, Im0, Re1, Im1, ...; ContainerType_Vector_LREAL if ipContour is of type ContainerType_Vector_TcVnPoint2_LREAL, else ContainerType_Vector_REAL.) *)
		nDescriptors	:	DINT;	(* Specifies how many descriptors should be returned (set to -1 to return all computed descriptors, i.e. at least as many as the number of contour points) *)
		hrPrev	:	HRESULT;	(* HRESULT indicating the result of previous operations (If SUCCEEDED(hrPrev) equals false, no operation is executed.) *)
	END_VAR

END_FUNCTION

// Functions/Contour Analysis/F_VN_MatchContours

	{attribute 'TcIecLibraryType'}
	{attribute 'external_name' := 'F_VN_MatchContours_GUID_E8C39366_6B22_DD46_88FA_6CF097A6F241'}
	(* Compare contours using the Hu moment invariants. In case of multiple contours in each container, the best matches are found and the average dissimilarity over all matched contours is returned. *)
	FUNCTION F_VN_MatchContours : HRESULT
	VAR_INPUT
		ipContour1	:	ITcVnContainer;	(* First contour (ContainerType_Vector_TcVnPoint2_DINT or ContainerType_Vector_TcVnPoint2_REAL; The elements of this container are the points of the contour) or collection of multiple contours (ContainerType_Vector_Vector_TcVnPoint2_DINT) *)
		ipContour2	:	ITcVnContainer;	(* Second contour (same type as ipContour1) *)
		eComparisonMethod	:	ETcVnContoursMatchComparisonMethod;	(* Method used for comparing the Hu moment invariants of the contours *)
	END_VAR
	VAR_IN_OUT
		fDissimilarity	:	LREAL;	(* Returns the dissimilarity of the contours depending on the chosen comparison method *)
	END_VAR
	VAR_INPUT
		hrPrev	:	HRESULT;	(* HRESULT indicating the result of previous operations (If SUCCEEDED(hrPrev) equals false, no operation is executed.) *)
	END_VAR

END_FUNCTION

// Functions/Contour Analysis/F_VN_MatchContoursExp

	{attribute 'TcIecLibraryType'}
	{attribute 'external_name' := 'F_VN_MatchContoursExp_GUID_99B8AA12_64AE_D55E_8E1B_0865B52A3A26'}
	(* Compare contours using the Hu moment invariants (and optionally further aspects). In case of multiple contours in each container, the best matches are found and the average dissimilarity over all matched contours is returned. (expert function) *)
	FUNCTION F_VN_MatchContoursExp : HRESULT
	VAR_INPUT
		ipContour1	:	ITcVnContainer;	(* First contour (ContainerType_Vector_TcVnPoint2_DINT or ContainerType_Vector_TcVnPoint2_REAL; The elements of this container are the points of the contour) or collection of multiple contours (ContainerType_Vector_Vector_TcVnPoint2_DINT) *)
		ipContour2	:	ITcVnContainer;	(* Second contour (same type as ipContour1) *)
		eComparisonMethod	:	ETcVnContoursMatchComparisonMethod;	(* Method used for comparing the Hu moment invariants of the contours *)
	END_VAR
	VAR_IN_OUT
		fDissimilarity	:	LREAL;	(* Returns the dissimilarity of the contours depending on the chosen comparison method *)
	END_VAR
	VAR_INPUT
		fAreaFactor	:	LREAL;	(* If > 0, the relative area difference between contours is scaled by this factor and added to the computed dissimilarity *)
		fAbsPositionFactor	:	LREAL;	(* If > 0, the absolute position difference between contours (i.e. the coordinates of the geometric contour centers) is scaled by this factor and added to the computed dissimilarity *)
		fRelPositionFactor	:	LREAL;	(* If > 0, the relative position difference between contours is scaled by this factor and added to the computed dissimilarity (only used if matching multiple contours) *)
		fNumDiffFactor	:	LREAL;	(* If > 0, the difference between the number of contours in both containers is scaled by this factor and added to the computed dissimilarity (only used if matching multiple contours) *)
		hrPrev	:	HRESULT;	(* HRESULT indicating the result of previous operations (If SUCCEEDED(hrPrev) equals false, no operation is executed.) *)
	END_VAR

END_FUNCTION

// Functions/Contour Analysis/F_VN_MatchContours1vsN

	{attribute 'TcIecLibraryType'}
	{attribute 'external_name' := 'F_VN_MatchContours1vsN_GUID_51F53F79_1BAD_D76C_BF22_8FB58CCC9364'}
	(* Compare a reference contour with multiple other contours using the Hu moment invariants. Returns a sorted list of best matches. *)
	FUNCTION F_VN_MatchContours1vsN : HRESULT
	VAR_INPUT
		ipRefContour	:	ITcVnContainer;	(* Reference contour (ContainerType_Vector_TcVnPoint2_DINT or ContainerType_Vector_TcVnPoint2_REAL; The elements of this container are the points of the contour) *)
		ipContours	:	ITcVnContainer;	(* Collection of multiple contours (CTcVnContainer_Vector_Vector_TcVnPoint2_DINT) *)
		ipMatchIndexes	:	REFERENCE TO ITcVnContainer;	(* Returns the indexes of the best matches (CTcVnContainer_Vector_ULINT; sorted, first element is best match, i.e. has lowest dissimilarity) *)
		ipDissimilarities	:	REFERENCE TO ITcVnContainer;	(* Returns the computed dissimilarities of the best matches (CTcVnContainer_Vector_LREAL; Optional, set to 0 if not required; sorted corresponding to ipMatchIndexes) *)
		fDissimilarityThreshold	:	LREAL;	(* Neglect irrelevant matches, i.e. dissimilarity > fDissimilarityThreshold *)
		eComparisonMethod	:	ETcVnContoursMatchComparisonMethod;	(* Method used for comparing the Hu moment invariants of the contours *)
		hrPrev	:	HRESULT;	(* HRESULT indicating the result of previous operations (If SUCCEEDED(hrPrev) equals false, no operation is executed.) *)
	END_VAR

END_FUNCTION

// Functions/Contour Analysis/F_VN_MatchContours1vsNExp

	{attribute 'TcIecLibraryType'}
	{attribute 'external_name' := 'F_VN_MatchContours1vsNExp_GUID_1CA1439C_95F5_DC65_8F25_ABAF19439829'}
	(* Compare a reference contour with multiple other contours using the Hu moment invariants (and optionally further aspects). Returns a sorted list of best matches. (expert function) *)
	FUNCTION F_VN_MatchContours1vsNExp : HRESULT
	VAR_INPUT
		ipRefContour	:	ITcVnContainer;	(* Reference contour (ContainerType_Vector_TcVnPoint2_DINT or ContainerType_Vector_TcVnPoint2_REAL; The elements of this container are the points of the contour) *)
		ipContours	:	ITcVnContainer;	(* Collection of multiple contours (CTcVnContainer_Vector_Vector_TcVnPoint2_DINT) *)
		ipMatchIndexes	:	REFERENCE TO ITcVnContainer;	(* Returns the indexes of the best matches (CTcVnContainer_Vector_ULINT; sorted, first element is best match, i.e. has lowest dissimilarity) *)
		ipDissimilarities	:	REFERENCE TO ITcVnContainer;	(* Returns the computed dissimilarities of the best matches (CTcVnContainer_Vector_LREAL; Optional, set to 0 if not required; sorted corresponding to ipMatchIndexes) *)
		fDissimilarityThreshold	:	LREAL;	(* Neglect irrelevant matches, i.e. dissimilarity > fDissimilarityThreshold *)
		eComparisonMethod	:	ETcVnContoursMatchComparisonMethod;	(* Method used for comparing the Hu moment invariants of the contours *)
		fAreaFactor	:	LREAL;	(* If > 0, the relative area difference between contours is scaled by this factor and added to the computed dissimilarity *)
		fAbsPositionFactor	:	LREAL;	(* If > 0, the absolute position difference between contours (i.e. the coordinates of the geometric contour centers) is scaled by this factor and added to the computed dissimilarity *)
		hrPrev	:	HRESULT;	(* HRESULT indicating the result of previous operations (If SUCCEEDED(hrPrev) equals false, no operation is executed.) *)
	END_VAR

END_FUNCTION

// Functions/Contour Analysis/F_VN_UprightBoundingRectangle

	{attribute 'TcIecLibraryType'}
	{attribute 'external_name' := 'F_VN_UprightBoundingRectangle_GUID_5F59B6C4_8783_DAD0_92AD_5F37DF8A0888'}
	(* Determines the upright bounding rectangle of a set of points. *)
	FUNCTION F_VN_UprightBoundingRectangle : HRESULT
	VAR_INPUT
		ipPointSet	:	ITcVnContainer;	(* Source point set (ContainerType_Vector_TcVnPoint2_DINT or ContainerType_Vector_TcVnPoint2_REAL; The elements of this container are the individual points.) *)
	END_VAR
	VAR_IN_OUT
		stRectangle	:	TcVnRectangle_UDINT;	(* Returns the determined rectangle *)
	END_VAR
	VAR_INPUT
		hrPrev	:	HRESULT;	(* HRESULT indicating the result of previous operations (If SUCCEEDED(hrPrev) equals false, no operation is executed.) *)
	END_VAR

END_FUNCTION

// Functions/Image Filtering/F_VN_BilateralFilter

	{attribute 'TcIecLibraryType'}
	{attribute 'external_name' := 'F_VN_BilateralFilter_GUID_6499BEA8_328C_DBFD_9EF7_B2759631EF92'}
	(* Apply a Bilateral filter to smooth the image but preserve edges. *)
	FUNCTION F_VN_BilateralFilter : HRESULT
	VAR_INPUT
		ipSrcImage	:	ITcVnImage;	(* Source image *)
		ipDestImage	:	REFERENCE TO ITcVnImage;	(* Destination image (Must be different from ipSrcImage! An appropriate destination image will be created if required.) *)
		nDiameter	:	DINT;	(* Diameter of the pixel neighborhood used for filtering (e.g. 5, 7, 9). If <= 0, it is automatically chosen dependend on fSigmaSpace. *)
		fSigmaColor	:	LREAL;	(* Sigma used for color space filtering (> 0). A larger value means that farther colors are mixed together. *)
		fSigmaSpace	:	LREAL;	(* Sigma used for coordinate space filtering (> 0). A larger value means that farther pixels can influence each other. *)
		hrPrev	:	HRESULT;	(* HRESULT indicating the result of previous operations (If SUCCEEDED(hrPrev) equals false, no operation is executed.) *)
	END_VAR

END_FUNCTION

// Functions/Image Filtering/F_VN_BilateralFilterExp

	{attribute 'TcIecLibraryType'}
	{attribute 'external_name' := 'F_VN_BilateralFilterExp_GUID_984FEB44_BA68_DD52_A7F8_59852AF41A51'}
	(* Apply a Bilateral filter to smooth the image but preserve edges. (expert function) *)
	FUNCTION F_VN_BilateralFilterExp : HRESULT
	VAR_INPUT
		ipSrcImage	:	ITcVnImage;	(* Source image *)
		ipDestImage	:	REFERENCE TO ITcVnImage;	(* Destination image (Must be different from ipSrcImage! An appropriate destination image will be created if required.) *)
		nDiameter	:	DINT;	(* Diameter of the pixel neighborhood used for filtering (e.g. 5, 7, 9). If <= 0, it is automatically chosen dependend on fSigmaSpace. *)
		fSigmaColor	:	LREAL;	(* Sigma used for color space filtering (> 0). A larger value means that farther colors are mixed together. *)
		fSigmaSpace	:	LREAL;	(* Sigma used for coordinate space filtering (> 0). A larger value means that farther pixels can influence each other. *)
		eBorderType	:	ETcVnBorderInterpolationMethod;	(* Image border handling *)
		hrPrev	:	HRESULT;	(* HRESULT indicating the result of previous operations (If SUCCEEDED(hrPrev) equals false, no operation is executed.) *)
	END_VAR

END_FUNCTION

// Functions/Image Filtering/F_VN_BoxFilter

	{attribute 'TcIecLibraryType'}
	{attribute 'external_name' := 'F_VN_BoxFilter_GUID_A3BB3964_6433_D078_9876_AD4E3C123067'}
	(* Apply a box filter to an image. *)
	FUNCTION F_VN_BoxFilter : HRESULT
	VAR_INPUT
		ipSrcImage	:	ITcVnImage;	(* Source image *)
		ipDestImage	:	REFERENCE TO ITcVnImage;	(* Destination image (An appropriate destination image will be created if required.) *)
		nFilterWidth	:	UDINT;	(* Filter width in pixels *)
		nFilterHeight	:	UDINT;	(* Filter height in pixels *)
		hrPrev	:	HRESULT;	(* HRESULT indicating the result of previous operations (If SUCCEEDED(hrPrev) equals false, no operation is executed.) *)
	END_VAR

END_FUNCTION

// Functions/Image Filtering/F_VN_BoxFilterExp

	{attribute 'TcIecLibraryType'}
	{attribute 'external_name' := 'F_VN_BoxFilterExp_GUID_FB19D2FE_8744_D70C_BECE_1D460FB06D5A'}
	(* Apply a box filter to an image. (expert function) *)
	FUNCTION F_VN_BoxFilterExp : HRESULT
	VAR_INPUT
		ipSrcImage	:	ITcVnImage;	(* Source image *)
		ipDestImage	:	REFERENCE TO ITcVnImage;	(* Destination image (An appropriate destination image will be created if required.) *)
		nFilterWidth	:	UDINT;	(* Filter width in pixels *)
		nFilterHeight	:	UDINT;	(* Filter height in pixels *)
		eDestDepth	:	ETcVnElementType;	(* Destination image depth *)
	END_VAR
	VAR_IN_OUT
		aAnchor	:	TcVnPoint;	(* Anchor point of the kernel ([-1, -1] for center) *)
	END_VAR
	VAR_INPUT
		bNormalize	:	BOOL;	(* If true, the kernel is normalized by nFilterWidth * nFilterHeight *)
		eBorderType	:	ETcVnBorderInterpolationMethod;	(* Image border handling *)
		hrPrev	:	HRESULT;	(* HRESULT indicating the result of previous operations (If SUCCEEDED(hrPrev) equals false, no operation is executed.) *)
	END_VAR

END_FUNCTION

// Functions/Image Filtering/F_VN_BrightBorderObjects

